# B&R Automation Studio project warcabot
Automation Studio 6.7.0.187; technology packages: mappCockpit 6.7.0, mappMotion 6.7.2, mappServices 6.7.1, mappView 6.7.0, mappVision 6.7.0, OpcUaCs 6.7.0

## Configuration Config1

CPU 5APC3100.KBU1-000, AutomationRuntime 6.7.6, Build 11.3.0

### Task classes (Cpu.sw)
```
Cyclic#4:
  Program <- Programs.Motion.Program.prg
  TestOpcua <- Programs.TestOpcua.prg
Libraries: McBase, MpRobotics, McAxGroup, McPathGen, MpAxis, runtime, CoTrace, McAxis, McAcpAx, McAcpPar, AsZip, FileIO, sys_lib, AsBrStr, MpBase, McProgInt, astime, ViBase, AsARCfg, powerlnk, AsEPL, AsIO, AsTCP, DataObj, ArSsl
```

### Hardware
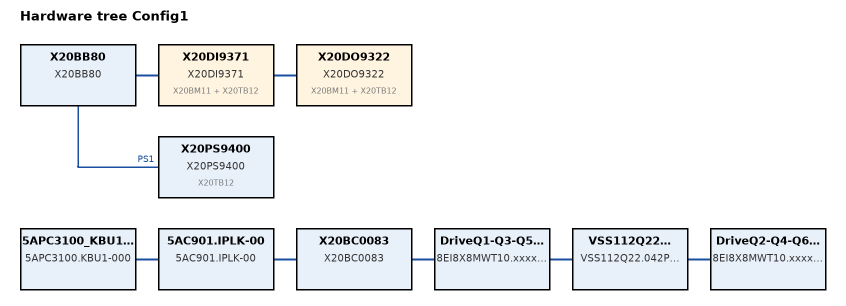
```
5AC901.IPLK-00 : 5AC901.IPLK-00 v2.1.0.0  [SL -> 5APC3100_KBU1_000.SL2]
  Connector IF1:
    MtuSize = 1500
    Channel1
    ChannelID1 = McAcpBroadcast
    ChannelType1 = OCTET[192]
    InternetAddress = 192.168.200.240
    SubnetMask = 255.255.255.0
  Supervision = off
5APC3100_KBU1_000 : 5APC3100.KBU1-000 v2.3.1.0
  Connector IF3:
    AssignedOperatingSystem = ARemb
    ActivateDevice = 1
    Mode = Manual
    InternetAddress = 192.168.0.11
    SubnetMask = 255.255.255.0
    ActivateSnmp = 2
  Connector IF4:
    AssignedOperatingSystem = ARemb
    ActivateDevice = 1
    Mode = DHCPServer
    InternetAddress = 192.168.1.11
    SubnetMask = 255.255.255.0
    Lease1
    LeaseName1 = Test
    LeaseStartAddress1 = 192.168.1.12
    LeaseStopAddress1 = 192.168.1.15
    LeaseSubnetMask1 = 255.255.255.0
    ActivateSnmp = 2
  Connector IF5:
    AssignedOperatingSystem = ARemb
  Connector IF6:
    AssignedOperatingSystem = ARemb
  Connector IF7:
    AssignedOperatingSystem = ARemb
  Connector IF8:
    AssignedOperatingSystem = ARemb
  ConfigurationID = warcabot_Config1
  Simulation = 1
  RemMemDevice = PCI.2.IPLK.SRAM
  RemMemSize = 1000
  PermanentPvSize = 500
  TimerDeviceType = EPLX2X
  TimerDevice = 5AC901.IPLK-00.IF1
  TaskClassIdleTime = 2000
  Cyclic1Duration = 2000
  Cyclic1Tolerance = 0
  FileDevice1
  FileDeviceName1 = USER
  FileDevicePath1 = USER_PATH
  FileDevice2
  FileDeviceName2 = CNC_PrgDir
  FileDevicePath2 = USER_PATH\Programs
  FileDevice3
  FileDeviceName3 = SG
  FileDevicePath3 = USER_PATH\SavedGames
  FileDevice4
  FileDeviceName4 = AH
  FileDevicePath4 = USER_PATH\AlarmHistory
  FileDevice5
  FileDeviceName5 = AUDIT
  FileDevicePath5 = USER_PATH\Audit
  FileDevice6
  FileDeviceName6 = REPORT
  FileDevicePath6 = USER_PATH\Report
  FileDevice7
  FileDeviceName7 = CF
  FileDevicePath7 = USER_PATH
  ActivateFtpServer = 1
  FtpAuthenticationType = FtpRoles
  FtpRole1
  FtpRoleName1 = Administraotr
  FTPRoleAccessRight1 = 0
  ActivateWebServer = 1
  WebServerProtocol = 1
  ActivateSdm = 1
  Authentication = 0
DriveQ1-Q3-Q5_Racer3_1 : 8EI8X8MWT10.xxxx-1 v2.4.0.0 (NodeNumber=2)  [PLK1 -> X20BC0083.PLK2 [Cable Type=PowerlinkCable, Length=10, Version=1.0.0.3]; PLK2 -> VSS112Q22.042P-000.PLK1 [Cable Type=PowerlinkCable, Length=10, Version=1.0.0.3]]
  DriveConfiguration/Encoder/EncoderX41:
    InterfaceType = EnDat
  DriveConfiguration/Encoder/EncoderX42:
    InterfaceType = EnDat
  DriveConfiguration/Encoder/EncoderX43:
    InterfaceType = EnDat
  DriveConfiguration/Channel[1]/RealAxis:
    AxisReference = gAxisQ1_Racer3_1
  DriveConfiguration/Channel[1]/RealAxis/MechanicalElements/Gearbox:
    Input = 81818
    Output = 1000
  DriveConfiguration/Channel[1]/RealAxis/MechanicalElements/RotaryToLinearTransformation:
    ReferenceDistance = 360
  DriveConfiguration/Channel[1]/RealAxis/Controller:
    Mode = PositionControllerWithTorqueFeedForward
  DriveConfiguration/Channel[1]/RealAxis/Controller/Mode/Position:
    ProportionalGain = 75
  DriveConfiguration/Channel[1]/RealAxis/Controller/Mode/Speed:
    FilterTime = 0.0008
  DriveConfiguration/Channel[1]/RealAxis/Controller/Mode:
    FeedForward = CyclicValueFromAxesGroup
  DriveConfiguration/Channel[1]/RealAxis/Homing:
    Mode = RestorePosition
    RestorePositionVariable = ::AxisRestorePos0
  DriveConfiguration/Channel[1]/RealAxis/MovementErrorLimits:
    PositionError = 1
  DriveConfiguration/Channel[1]/RealAxis:
    JerkFilter = Used
  DriveConfiguration/Channel[1]/RealAxis/JerkFilter:
    JerkTime = 0.01
  DriveConfiguration/Channel[1]/RealAxis/AxisFeatures:
    FeatureRef[1] = Feature_Brake_Racer3_1
  DriveConfiguration/Channel[2]/RealAxis:
    AxisReference = gAxisQ3_Racer3_1
  DriveConfiguration/Channel[2]/RealAxis/MechanicalElements/Gearbox:
    Input = 72
  DriveConfiguration/Channel[2]/RealAxis/MechanicalElements/RotaryToLinearTransformation:
    ReferenceDistance = 360
  DriveConfiguration/Channel[2]/RealAxis/Controller:
    Mode = PositionControllerWithTorqueFeedForward
  DriveConfiguration/Channel[2]/RealAxis/Controller/Mode/Speed:
    ProportionalGain = 1.5
    FilterTime = 0.0008
  DriveConfiguration/Channel[2]/RealAxis/Controller/Mode:
    FeedForward = CyclicValueFromAxesGroup
  DriveConfiguration/Channel[2]/RealAxis/Homing:
    Mode = RestorePosition
    RestorePositionVariable = ::AxisRestorePos2
  DriveConfiguration/Channel[2]/RealAxis/MovementErrorLimits:
    PositionError = 1
  DriveConfiguration/Channel[2]/RealAxis:
    JerkFilter = Used
  DriveConfiguration/Channel[2]/RealAxis/JerkFilter:
    JerkTime = 0.01
  DriveConfiguration/Channel[2]/RealAxis/AxisFeatures:
    FeatureRef[1] = Feature_Brake_Racer3_1
  DriveConfiguration/Channel[3]/RealAxis:
    AxisReference = gAxisQ5_Racer3_1
  DriveConfiguration/Channel[3]/RealAxis/MechanicalElements/Gearbox:
    Input = 612
    Output = 10
  DriveConfiguration/Channel[3]/RealAxis/MechanicalElements/RotaryToLinearTransformation:
    ReferenceDistance = 360
  DriveConfiguration/Channel[3]/RealAxis/Controller:
    Mode = PositionControllerWithTorqueFeedForward
  DriveConfiguration/Channel[3]/RealAxis/Controller/Mode/Position:
    ProportionalGain = 200
  DriveConfiguration/Channel[3]/RealAxis/Controller/Mode/Speed:
    ProportionalGain = 1.5
    FilterTime = 0.0008
  DriveConfiguration/Channel[3]/RealAxis/Controller/Mode:
    FeedForward = CyclicValueFromAxesGroup
  DriveConfiguration/Channel[3]/RealAxis/Homing:
    Mode = RestorePosition
    RestorePositionVariable = ::AxisRestorePos4
  DriveConfiguration/Channel[3]/RealAxis/MovementErrorLimits:
    PositionError = 1
  DriveConfiguration/Channel[3]/RealAxis:
    JerkFilter = Used
  DriveConfiguration/Channel[3]/RealAxis/JerkFilter:
    JerkTime = 0.01
  DriveConfiguration/Channel[3]/RealAxis/AxisFeatures:
    FeatureRef[1] = Feature_Brake_Racer3_1
DriveQ2-Q4-Q6_Racer3_1 : 8EI8X8MWT10.xxxx-1 v2.4.0.0 (NodeNumber=3)  [PLK1 -> VSS112Q22.042P-000.PLK2 [Cable Type=PowerlinkCable, Length=10, Version=1.0.0.3]]
  DriveConfiguration/Encoder/EncoderX41:
    InterfaceType = EnDat
  DriveConfiguration/Encoder/EncoderX42:
    InterfaceType = EnDat
  DriveConfiguration/Encoder/EncoderX43:
    InterfaceType = EnDat
  DriveConfiguration/Channel[1]/RealAxis:
    AxisReference = gAxisQ2_Racer3_1
  DriveConfiguration/Channel[1]/RealAxis/MechanicalElements/Gearbox:
    Input = 80
  DriveConfiguration/Channel[1]/RealAxis/MechanicalElements/RotaryToLinearTransformation:
    ReferenceDistance = 360
  DriveConfiguration/Channel[1]/RealAxis/Controller:
    Mode = PositionControllerWithTorqueFeedForward
  DriveConfiguration/Channel[1]/RealAxis/Controller/Mode/Speed:
    FilterTime = 0.0008
  DriveConfiguration/Channel[1]/RealAxis/Controller/Mode:
    FeedForward = CyclicValueFromAxesGroup
  DriveConfiguration/Channel[1]/RealAxis/Homing:
    Mode = RestorePosition
    RestorePositionVariable = ::AxisRestorePos1
  DriveConfiguration/Channel[1]/RealAxis/MovementErrorLimits:
    PositionError = 1
  DriveConfiguration/Channel[1]/RealAxis:
    JerkFilter = Used
  DriveConfiguration/Channel[1]/RealAxis/JerkFilter:
    JerkTime = 0.01
  DriveConfiguration/Channel[1]/RealAxis/AxisFeatures:
    FeatureRef[1] = Feature_Brake_Racer3_1
  DriveConfiguration/Channel[2]/RealAxis:
    AxisReference = gAxisQ4_Racer3_1
  DriveConfiguration/Channel[2]/RealAxis/MechanicalElements/Gearbox:
    Input = 612
    Output = 10
  DriveConfiguration/Channel[2]/RealAxis/MechanicalElements/RotaryToLinearTransformation:
    ReferenceDistance = 360
  DriveConfiguration/Channel[2]/RealAxis/Controller:
    Mode = PositionControllerWithTorqueFeedForward
  DriveConfiguration/Channel[2]/RealAxis/Controller/Mode/Position:
    ProportionalGain = 100
  DriveConfiguration/Channel[2]/RealAxis/Controller/Mode/Speed:
    FilterTime = 0.0008
  DriveConfiguration/Channel[2]/RealAxis/Controller/Mode:
    FeedForward = CyclicValueFromAxesGroup
  DriveConfiguration/Channel[2]/RealAxis/Homing:
    Mode = RestorePosition
    RestorePositionVariable = ::AxisRestorePos3
  DriveConfiguration/Channel[2]/RealAxis/MovementErrorLimits:
    PositionError = 1
  DriveConfiguration/Channel[2]/RealAxis:
    JerkFilter = Used
  DriveConfiguration/Channel[2]/RealAxis/JerkFilter:
    JerkTime = 0.01
  DriveConfiguration/Channel[2]/RealAxis/AxisFeatures:
    FeatureRef[1] = Feature_Brake_Racer3_1
  DriveConfiguration/Channel[3]/RealAxis:
    AxisReference = gAxisQ6_Racer3_1
  DriveConfiguration/Channel[3]/RealAxis/MechanicalElements/Gearbox:
    Input = 40
  DriveConfiguration/Channel[3]/RealAxis/MechanicalElements/RotaryToLinearTransformation:
    ReferenceDistance = 360
  DriveConfiguration/Channel[3]/RealAxis/Controller:
    Mode = PositionControllerWithTorqueFeedForward
  DriveConfiguration/Channel[3]/RealAxis/Controller/Mode/Position:
    ProportionalGain = 200
  DriveConfiguration/Channel[3]/RealAxis/Controller/Mode/Speed:
    ProportionalGain = 1.5
    FilterTime = 0.0008
  DriveConfiguration/Channel[3]/RealAxis/Controller/Mode:
    FeedForward = CyclicValueFromAxesGroup
  DriveConfiguration/Channel[3]/RealAxis/Homing:
    Mode = RestorePosition
    RestorePositionVariable = ::AxisRestorePos5
  DriveConfiguration/Channel[3]/RealAxis/MovementErrorLimits:
    PositionError = 1
  DriveConfiguration/Channel[3]/RealAxis:
    JerkFilter = Used
  DriveConfiguration/Channel[3]/RealAxis/JerkFilter:
    JerkTime = 0.01
  DriveConfiguration/Channel[3]/RealAxis/AxisFeatures:
    FeatureRef[1] = Feature_Brake_Racer3_1
VSS112Q22.042P-000 : VSS112Q22.042P-000 v1.11.0.929 (NodeNumber=4)  [PLK1 -> DriveQ1-Q3-Q5_Racer3_1.PLK2 [Cable Type=PowerlinkCable, Length=10, Version=1.0.0.3]; PLK2 -> DriveQ2-Q4-Q6_Racer3_1.PLK1 [Cable Type=PowerlinkCable, Length=10, Version=1.0.0.3]]
  VisionConfig = gCamera
X20BB80 : X20BB80 v1.1.0.0
X20BC0083 : X20BC0083 v2.17.0.0 (NodeNumber=1)  [PLK1 -> 5AC901.IPLK-00.IF1 [Cable Type=PowerlinkCable, Length=10, Version=1.0.0.3]; PLK2 -> DriveQ1-Q3-Q5_Racer3_1.PLK1 [Cable Type=PowerlinkCable, Length=10, Version=1.0.0.3]; SL -> X20BB80.SL1]
X20BM11 : X20BM11 v1.1.0.0  [X2X1 -> X20BB80.IF1]
X20BM11_a : X20BM11 v1.1.0.0  [X2X1 -> X20BM11.X2X2]
X20DI9371 : X20DI9371 v1.6.1.0  [SS1 -> X20TB12.SS; SL -> X20BM11.SL1]
X20DO9322 : X20DO9322 v1.7.0.0  [SS1 -> X20TB12_b.SS; SL -> X20BM11_a.SL1]
X20PS9400 : X20PS9400 v1.9.0.0  [SS1 -> X20TB12_a.SS; PS -> X20BB80.PS1]
X20TB12 : X20TB12 v1.0.0.0
X20TB12_a : X20TB12 v1.0.0.0
X20TB12_b : X20TB12 v1.0.0.0
```

### Cpu.per - 5APC3100_KBU1_000/Cpu.per
```iecst
VAR_CONFIG
	AxisRestorePos0 AT %M0; (* *)
	AxisRestorePos1 AT %M72; (* *)
	AxisRestorePos2 AT %M144; (* *)
	AxisRestorePos3 AT %M216; (* *)
	AxisRestorePos4 AT %M288; (* *)
	AxisRestorePos5 AT %M360; (* *)
END_VAR
```

### IoMap.iom - 5APC3100_KBU1_000/IoMap.iom
```iecst
VAR_CONFIG
	::Program2:gCameraCtrl.Cmd.AcquireImage AT %QX."VSS112Q22.042P-000".ImageAcquisition;
	::Program2:gCameraCtrl.Status.AcquisitionReady AT %IX."VSS112Q22.042P-000".ImageAcquisitionReady;
	::Program2:gCameraCtrl.Status.ProcessingError AT %IW."VSS112Q22.042P-000".ImageProcessingError;
	::Program2:gCameraCtrl.Status.ProcessingActive AT %IX."VSS112Q22.042P-000".ImageProcessingActive;
	::gCameraAutoAdjust AT %QX."VSS112Q22.042P-000".SearchAcquisitionSettings;
	::Program2:gCameraCtrl.Status.ReadFocus AT %IW."VSS112Q22.042P-000".ReadFocus;
	::Program2:gCameraCtrl.NumResults AT %IB."VSS112Q22.042P-000".NumResults_Out_1;
	::Program2:gCameraCtrl.Pieces[1].PositionX AT %ID."VSS112Q22.042P-000".PositionX_Out_101;
	::Program2:gCameraCtrl.Pieces[1].PositionY AT %ID."VSS112Q22.042P-000".PositionY_Out_101;
	::Program2:gCameraCtrl.Pieces[1].Area AT %ID."VSS112Q22.042P-000".Area_Out_101;
	::Program2:gCameraCtrl.Pieces[1].Score AT %IB."VSS112Q22.042P-000".Score_Out_101;
	::Program2:gCameraCtrl.Cmd.Enable AT %QX."VSS112Q22.042P-000".Enable_In_1;
	::Program2:gCameraCtrl.Pieces[1].ModelNumber AT %IB."VSS112Q22.042P-000".ModelNumber_Out_101;
	::Program2:gCameraCtrl.Parameters.NumSearchMax AT %QB."VSS112Q22.042P-000".NumSearchMax_In_1;
	::Program2:gCameraCtrl.Status.ReadExposureTime AT %ID."VSS112Q22.042P-000".ReadExposureTime;
	::Program2:gCameraCtrl.Pieces[2].ModelNumber AT %IB."VSS112Q22.042P-000".ModelNumber_Out_102;
	::Program2:gCameraCtrl.Pieces[2].Score AT %IB."VSS112Q22.042P-000".Score_Out_102;
	::Program2:gCameraCtrl.Pieces[2].PositionX AT %ID."VSS112Q22.042P-000".PositionX_Out_102;
	::Program2:gCameraCtrl.Pieces[2].PositionY AT %ID."VSS112Q22.042P-000".PositionY_Out_102;
	::Program2:gCameraCtrl.Pieces[3].ModelNumber AT %IB."VSS112Q22.042P-000".ModelNumber_Out_103;
	::Program2:gCameraCtrl.Pieces[3].Score AT %IB."VSS112Q22.042P-000".Score_Out_103;
	::Program2:gCameraCtrl.Pieces[3].PositionX AT %ID."VSS112Q22.042P-000".PositionX_Out_103;
	::Program2:gCameraCtrl.Pieces[3].PositionY AT %ID."VSS112Q22.042P-000".PositionY_Out_103;
	::Program2:gCameraCtrl.Pieces[4].ModelNumber AT %IB."VSS112Q22.042P-000".ModelNumber_Out_104;
	::Program2:gCameraCtrl.Pieces[5].ModelNumber AT %IB."VSS112Q22.042P-000".ModelNumber_Out_105;
	::Program2:gCameraCtrl.Pieces[6].ModelNumber AT %IB."VSS112Q22.042P-000".ModelNumber_Out_106;
	::Program2:gCameraCtrl.Pieces[7].ModelNumber AT %IB."VSS112Q22.042P-000".ModelNumber_Out_107;
	::Program2:gCameraCtrl.Pieces[8].ModelNumber AT %IB."VSS112Q22.042P-000".ModelNumber_Out_108;
	::Program2:gCameraCtrl.Pieces[9].ModelNumber AT %IB."VSS112Q22.042P-000".ModelNumber_Out_109;
	::Program2:gCameraCtrl.Pieces[10].ModelNumber AT %IB."VSS112Q22.042P-000".ModelNumber_Out_110;
	::Program2:gCameraCtrl.Pieces[11].ModelNumber AT %IB."VSS112Q22.042P-000".ModelNumber_Out_111;
	::Program2:gCameraCtrl.Pieces[12].ModelNumber AT %IB."VSS112Q22.042P-000".ModelNumber_Out_112;
	::Program2:gCameraCtrl.Pieces[13].ModelNumber AT %IB."VSS112Q22.042P-000".ModelNumber_Out_113;
	::Program2:gCameraCtrl.Pieces[14].ModelNumber AT %IB."VSS112Q22.042P-000".ModelNumber_Out_114;
	::Program2:gCameraCtrl.Pieces[15].ModelNumber AT %IB."VSS112Q22.042P-000".ModelNumber_Out_115;
	::Program2:gCameraCtrl.Pieces[16].ModelNumber AT %IB."VSS112Q22.042P-000".ModelNumber_Out_116;
	::Program2:gCameraCtrl.Pieces[17].ModelNumber AT %IB."VSS112Q22.042P-000".ModelNumber_Out_117;
	::Program2:gCameraCtrl.Pieces[18].ModelNumber AT %IB."VSS112Q22.042P-000".ModelNumber_Out_118;
	::Program2:gCameraCtrl.Pieces[19].ModelNumber AT %IB."VSS112Q22.042P-000".ModelNumber_Out_119;
	::Program2:gCameraCtrl.Pieces[20].ModelNumber AT %IB."VSS112Q22.042P-000".ModelNumber_Out_120;
	::Program2:gCameraCtrl.Pieces[21].ModelNumber AT %IB."VSS112Q22.042P-000".ModelNumber_Out_121;
	::Program2:gCameraCtrl.Pieces[22].ModelNumber AT %IB."VSS112Q22.042P-000".ModelNumber_Out_122;
	::Program2:gCameraCtrl.Pieces[23].ModelNumber AT %IB."VSS112Q22.042P-000".ModelNumber_Out_123;
	::Program2:gCameraCtrl.Pieces[24].ModelNumber AT %IB."VSS112Q22.042P-000".ModelNumber_Out_124;
	::Program2:gCameraCtrl.Pieces[4].Score AT %IB."VSS112Q22.042P-000".Score_Out_104;
	::Program2:gCameraCtrl.Pieces[5].Score AT %IB."VSS112Q22.042P-000".Score_Out_105;
	::Program2:gCameraCtrl.Pieces[6].Score AT %IB."VSS112Q22.042P-000".Score_Out_106;
	::Program2:gCameraCtrl.Pieces[7].Score AT %IB."VSS112Q22.042P-000".Score_Out_107;
	::Program2:gCameraCtrl.Pieces[8].Score AT %IB."VSS112Q22.042P-000".Score_Out_108;
	::Program2:gCameraCtrl.Pieces[9].Score AT %IB."VSS112Q22.042P-000".Score_Out_109;
	::Program2:gCameraCtrl.Pieces[10].Score AT %IB."VSS112Q22.042P-000".Score_Out_110;
	::Program2:gCameraCtrl.Pieces[11].Score AT %IB."VSS112Q22.042P-000".Score_Out_111;
	::Program2:gCameraCtrl.Pieces[12].Score AT %IB."VSS112Q22.042P-000".Score_Out_112;
	::Program2:gCameraCtrl.Pieces[13].Score AT %IB."VSS112Q22.042P-000".Score_Out_113;
	::Program2:gCameraCtrl.Pieces[14].Score AT %IB."VSS112Q22.042P-000".Score_Out_114;
	::Program2:gCameraCtrl.Pieces[15].Score AT %IB."VSS112Q22.042P-000".Score_Out_115;
	::Program2:gCameraCtrl.Pieces[16].Score AT %IB."VSS112Q22.042P-000".Score_Out_116;
	::Program2:gCameraCtrl.Pieces[17].Score AT %IB."VSS112Q22.042P-000".Score_Out_117;
	::Program2:gCameraCtrl.Pieces[18].Score AT %IB."VSS112Q22.042P-000".Score_Out_118;
	::Program2:gCameraCtrl.Pieces[19].Score AT %IB."VSS112Q22.042P-000".Score_Out_119;
	::Program2:gCameraCtrl.Pieces[20].Score AT %IB."VSS112Q22.042P-000".Score_Out_120;
	::Program2:gCameraCtrl.Pieces[21].Score AT %IB."VSS112Q22.042P-000".Score_Out_121;
	::Program2:gCameraCtrl.Pieces[22].Score AT %IB."VSS112Q22.042P-000".Score_Out_122;
	::Program2:gCameraCtrl.Pieces[23].Score AT %IB."VSS112Q22.042P-000".Score_Out_123;
	::Program2:gCameraCtrl.Pieces[24].Score AT %IB."VSS112Q22.042P-000".Score_Out_124;
	::Program2:gCameraCtrl.Pieces[4].PositionX AT %ID."VSS112Q22.042P-000".PositionX_Out_104;
	::Program2:gCameraCtrl.Pieces[5].PositionX AT %ID."VSS112Q22.042P-000".PositionX_Out_105;
	::Program2:gCameraCtrl.Pieces[6].PositionX AT %ID."VSS112Q22.042P-000".PositionX_Out_106;
	::Program2:gCameraCtrl.Pieces[7].PositionX AT %ID."VSS112Q22.042P-000".PositionX_Out_107;
	::Program2:gCameraCtrl.Pieces[8].PositionX AT %ID."VSS112Q22.042P-000".PositionX_Out_108;
	::Program2:gCameraCtrl.Pieces[9].PositionX AT %ID."VSS112Q22.042P-000".PositionX_Out_109;
	::Program2:gCameraCtrl.Pieces[10].PositionX AT %ID."VSS112Q22.042P-000".PositionX_Out_110;
	::Program2:gCameraCtrl.Pieces[11].PositionX AT %ID."VSS112Q22.042P-000".PositionX_Out_111;
	::Program2:gCameraCtrl.Pieces[12].PositionX AT %ID."VSS112Q22.042P-000".PositionX_Out_112;
	::Program2:gCameraCtrl.Pieces[13].PositionX AT %ID."VSS112Q22.042P-000".PositionX_Out_113;
	::Program2:gCameraCtrl.Pieces[14].PositionX AT %ID."VSS112Q22.042P-000".PositionX_Out_114;
	::Program2:gCameraCtrl.Pieces[15].PositionX AT %ID."VSS112Q22.042P-000".PositionX_Out_115;
	::Program2:gCameraCtrl.Pieces[16].PositionX AT %ID."VSS112Q22.042P-000".PositionX_Out_116;
	::Program2:gCameraCtrl.Pieces[17].PositionX AT %ID."VSS112Q22.042P-000".PositionX_Out_117;
	::Program2:gCameraCtrl.Pieces[18].PositionX AT %ID."VSS112Q22.042P-000".PositionX_Out_118;
	::Program2:gCameraCtrl.Pieces[19].PositionX AT %ID."VSS112Q22.042P-000".PositionX_Out_119;
	::Program2:gCameraCtrl.Pieces[20].PositionX AT %ID."VSS112Q22.042P-000".PositionX_Out_120;
	::Program2:gCameraCtrl.Pieces[21].PositionX AT %ID."VSS112Q22.042P-000".PositionX_Out_121;
	::Program2:gCameraCtrl.Pieces[22].PositionX AT %ID."VSS112Q22.042P-000".PositionX_Out_122;
	::Program2:gCameraCtrl.Pieces[23].PositionX AT %ID."VSS112Q22.042P-000".PositionX_Out_123;
	::Program2:gCameraCtrl.Pieces[24].PositionX AT %ID."VSS112Q22.042P-000".PositionX_Out_124;
	::Program2:gCameraCtrl.Pieces[4].PositionY AT %ID."VSS112Q22.042P-000".PositionY_Out_104;
	::Program2:gCameraCtrl.Pieces[5].PositionY AT %ID."VSS112Q22.042P-000".PositionY_Out_105;
	::Program2:gCameraCtrl.Pieces[6].PositionY AT %ID."VSS112Q22.042P-000".PositionY_Out_106;
	::Program2:gCameraCtrl.Pieces[7].PositionY AT %ID."VSS112Q22.042P-000".PositionY_Out_107;
	::Program2:gCameraCtrl.Pieces[8].PositionY AT %ID."VSS112Q22.042P-000".PositionY_Out_108;
	::Program2:gCameraCtrl.Pieces[9].PositionY AT %ID."VSS112Q22.042P-000".PositionY_Out_109;
	::Program2:gCameraCtrl.Pieces[10].PositionY AT %ID."VSS112Q22.042P-000".PositionY_Out_110;
	::Program2:gCameraCtrl.Pieces[11].PositionY AT %ID."VSS112Q22.042P-000".PositionY_Out_111;
	::Program2:gCameraCtrl.Pieces[12].PositionY AT %ID."VSS112Q22.042P-000".PositionY_Out_112;
	::Program2:gCameraCtrl.Pieces[13].PositionY AT %ID."VSS112Q22.042P-000".PositionY_Out_113;
	::Program2:gCameraCtrl.Pieces[14].PositionY AT %ID."VSS112Q22.042P-000".PositionY_Out_114;
	::Program2:gCameraCtrl.Pieces[15].PositionY AT %ID."VSS112Q22.042P-000".PositionY_Out_115;
	::Program2:gCameraCtrl.Pieces[16].PositionY AT %ID."VSS112Q22.042P-000".PositionY_Out_116;
	::Program2:gCameraCtrl.Pieces[17].PositionY AT %ID."VSS112Q22.042P-000".PositionY_Out_117;
	::Program2:gCameraCtrl.Pieces[18].PositionY AT %ID."VSS112Q22.042P-000".PositionY_Out_118;
	::Program2:gCameraCtrl.Pieces[19].PositionY AT %ID."VSS112Q22.042P-000".PositionY_Out_119;
	::Program2:gCameraCtrl.Pieces[20].PositionY AT %ID."VSS112Q22.042P-000".PositionY_Out_120;
	::Program2:gCameraCtrl.Pieces[21].PositionY AT %ID."VSS112Q22.042P-000".PositionY_Out_121;
	::Program2:gCameraCtrl.Pieces[22].PositionY AT %ID."VSS112Q22.042P-000".PositionY_Out_122;
	::Program2:gCameraCtrl.Pieces[23].PositionY AT %ID."VSS112Q22.042P-000".PositionY_Out_123;
	::Program2:gCameraCtrl.Pieces[24].PositionY AT %ID."VSS112Q22.042P-000".PositionY_Out_124;
	Cyclic#1.::doMagnet AT %QX."X20DO9322".DigitalOutput05;
	::Program2:gCameraCtrl.Parameters.ExposureTime AT %QD."VSS112Q22.042P-000".ExposureTime01;
	::Program2:gCameraCtrl.Parameters.SetFocus AT %QW."VSS112Q22.042P-000".SetFocus;
	::Program2:gCameraCtrl.Parameters.GainLevel AT %QB."VSS112Q22.042P-000".GainLevel;
	::Program2:gCameraCtrl.Status.ReadGainLevel AT %IB."VSS112Q22.042P-000".ReadGainLevel;
	::Program2:gCameraCtrl.Pieces[25].ModelNumber AT %IB."VSS112Q22.042P-000".ModelNumber_Out_125;
	::Program2:gCameraCtrl.Pieces[26].ModelNumber AT %IB."VSS112Q22.042P-000".ModelNumber_Out_126;
	::Program2:gCameraCtrl.Pieces[25].Score AT %IB."VSS112Q22.042P-000".Score_Out_125;
	::Program2:gCameraCtrl.Pieces[26].Score AT %IB."VSS112Q22.042P-000".Score_Out_126;
	::Program2:gCameraCtrl.Pieces[25].PositionX AT %ID."VSS112Q22.042P-000".PositionX_Out_125;
	::Program2:gCameraCtrl.Pieces[26].PositionX AT %ID."VSS112Q22.042P-000".PositionX_Out_126;
	::Program2:gCameraCtrl.Pieces[25].PositionY AT %ID."VSS112Q22.042P-000".PositionY_Out_125;
	::Program2:gCameraCtrl.Pieces[26].PositionY AT %ID."VSS112Q22.042P-000".PositionY_Out_126;
	::Program2:gCameraCtrl.Parameters.FlashColor AT %QB."VSS112Q22.042P-000".FlashColor01;
	::Program2:gCameraCtrl.Parameters.FlashSegment AT %QB."VSS112Q22.042P-000".FlashSegment01;
END_VAR
```

### GroupConf.axesgroup - 5APC3100_KBU1_000/mappMotion/6AxesRoboArmA/GroupConf.axesgroup
```
Element gAxesGroup_Racer3_1 (Type=axesgroup)
  Type = PathGenAxesGroup
    PhysicalAxes:
      JointAxes:
        JointAxis[1]:
          AxisRef = gAxisQ1_Racer3_1
        JointAxis[2]:
          AxisRef = gAxisQ2_Racer3_1
        JointAxis[3]:
          AxisRef = gAxisQ3_Racer3_1
        JointAxis[4]:
          AxisRef = gAxisQ4_Racer3_1
        JointAxis[5]:
          AxisRef = gAxisQ5_Racer3_1
        JointAxis[6]:
          AxisRef = gAxisQ6_Racer3_1
    MechanicalSystem:
      MechSysRef = MechSys_Racer3_1
    BasicSettings:
      GeometryPlanning:
        MaxTangentialTransitionDeviation = 0.05
      TrajectoryPlanning:
        LimitCheckResolution:
          Time = 0.005
        BufferTime:
          Time = 0.050
    AxesGroupFeatures:
      FeatureRef[1] = Feature_Programs_Racer3_1
      FeatureRef[2] = Feature_FeedForward_Racer3_1
      FeatureRef[3] = Feature_Jogging_Racer3_1
      FeatureRef[4] = Feature_SharedBrakesSignals_Racer3_1
      FeatureRef[5] = Feature_WorkspaceMonitoring_Racer3_1
```

### GroupFeat.axesgroupfeature - 5APC3100_KBU1_000/mappMotion/6AxesRoboArmA/GroupFeat.axesgroupfeature
```
Element Feature_Programs_Racer3_1 (Type=axesgroupfeature)
Element Feature_FeedForward_Racer3_1 (Type=axesgroupfeature)
  Type = FeedForward
    RiseTime = 0.25
Element Feature_Jogging_Racer3_1 (Type=axesgroupfeature)
  Type = Jogging
Element Feature_SharedBrakesSignals_Racer3_1 (Type=axesgroupfeature)
  Type = SharedBrakesSignals
    BrakeComposite[1]:
      Axes:
        AxisRef[1] = gAxisQ1_Racer3_1
        AxisRef[2] = gAxisQ2_Racer3_1
        AxisRef[3] = gAxisQ3_Racer3_1
      Output:
        AxisRef = gAxisQ1_Racer3_1
    BrakeComposite[2]:
      Axes:
        AxisRef[1] = gAxisQ4_Racer3_1
        AxisRef[2] = gAxisQ5_Racer3_1
        AxisRef[3] = gAxisQ6_Racer3_1
      Output:
        AxisRef = gAxisQ4_Racer3_1
Element Feature_WorkspaceMonitoring_Racer3_1 (Type=axesgroupfeature)
  Type = WorkspaceMonitoring
    WorkspaceRef = Workspace_1
    SelfCollisionDetection = Enabled
Element Feature_Monitoring_Racer3_2 (Type=axesgroupfeature)
  Type = MonitoringElements
    SingleElements:
      SingleElement[1] = WorkspaceMonitoring
        Level = ::WorkspaceMonitor
```

### MechSys.mechanicalsystem - 5APC3100_KBU1_000/mappMotion/6AxesRoboArmA/MechSys.mechanicalsystem
```
Element MechSys_Racer3_1 (Type=mechanicalsystem)
  Type = 6AxesRoboarm
    Subtype = 6AxesRoboarmB
      Description:
        Dimensions:
          TranslationFromBaseToQ1IsReadOnly = 1
          TranslationFromQ1ToQ2IsReadOnly = 1
          TranslationFromQ1ToQ2:
            X = 50.0
            Z = 365.0
          TranslationFromQ2ToQ3IsReadOnly = 1
          TranslationFromQ2ToQ3:
            Z = 270.0
          TranslationFromQ3ToQ4IsReadOnly = 1
          TranslationFromQ3ToQ4:
            X = -50.0
          TranslationFromQ4ToQ5IsReadOnly = 1
          TranslationFromQ4ToQ5:
            Z = 305.94
          TranslationFromQ5ToQ6IsReadOnly = 1
          TranslationFromQ6ToFlange:
            Z = 120
        Offsets:
          JointAxisIsReadOnly = 1
          JointAxis[1]
          JointAxis[2]
          JointAxis[3]
          JointAxis[4]
          JointAxis[5]
          JointAxis[6]
        CountDirections:
          JointAxisIsReadOnly = 1
          JointAxis[1] = Inverse
          JointAxis[2]
          JointAxis[3] = Inverse
          JointAxis[4] = Inverse
          JointAxis[5]
          JointAxis[6] = Inverse
      InternalDynamicModel = Used
        TypeIsReadOnly = 1
        Type = Comau Racer 3
        Row[1]:
          Value = 4
          Unit = 
          Description = TRF_DYN11D_typ
        Row[2]:
          Index = 1
          Value = 0
          Unit = 
          Description = 
        Row[3]:
          Index = 2
          Value = 0
          Unit = 
          Description = 
        Row[4]:
          Index = 3
          Value = 0.99502
          Unit = kgm^2
          Description = m1*rc1x^2+m1*rc1y^2+Jzz1+(0.0025)*m2+m2*rc2y^2+(0.5)*Jxx2+(-0.5)*Jyy2+(0.5)*Jzz2+(0.0025)*m3+m3*rc3y^2+(0.5)*Jxx3+(-0.5)*Jyy3+(0.5)*Jzz3+(0.0025)*m4+(0.0025)*m5+(0.0025)*m6+(6694.1851)*JDrive1+(-3200)*JDrive2
        Row[5]:
          Index = 4
          Value = 0
          Unit = 
          Description = 
        Row[6]:
          Index = 5
          Value = 0
          Unit = 
          Description = 
        Row[7]:
          Index = 6
          Value = 0
          Unit = 
          Description = 
        Row[8]:
          Index = 7
          Value = -0.0079739
          Unit = kgm
          Description = m2*rc2x
        Row[9]:
          Index = 8
          Value = 0
          Unit = 
          Description = 
        Row[10]:
          Index = 9
          Value = 3.2569
          Unit = kgm
          Description = m2*rc2z+(0.27)*m3+(0.27)*m4+(0.27)*m5+(0.27)*m6
        Row[11]:
          Index = 10
          Value = -0.01529
          Unit = kgm^2
          Description = m2*rc2x*rc2y
        Row[12]:
          Index = 11
          Value = 0.018218
          Unit = kgm^2
          Description = m2*rc2y*rc2z+(0.27)*m3*rc3y
        Row[13]:
          Index = 12
          Value = -0.027
          Unit = kgm^2
          Description = m2*rc2x*rc2z
        Row[14]:
          Index = 13
          Value = 0.23153
          Unit = kgm^2
          Description = m2*rc2x^2+(-0.5)*Jxx2+(0.5)*Jyy2+(0.5)*Jzz2+(3200)*JDrive2
        Row[15]:
          Index = 14
          Value = 0
          Unit = 
          Description = 
        Row[16]:
          Index = 15
          Value = 1.1014
          Unit = kgm^2
          Description = m2*rc2z^2+(0.5)*Jxx2+(0.5)*Jyy2+(-0.5)*Jzz2+(0.0729)*m3+(0.0729)*m4+(0.0729)*m5+(0.0729)*m6+(3200)*JDrive2
        Row[17]:
          Index = 16
          Value = 0
          Unit = 
          Description = 
        Row[18]:
          Index = 17
          Value = 0
          Unit = 
          Description = 
        Row[19]:
          Index = 18
          Value = 0
          Unit = 
          Description = 
        Row[20]:
          Index = 19
          Value = 0
          Unit = 
          Description = 
        Row[21]:
          Index = 20
          Value = -0.32261
          Unit = kgm
          Description = m3*rc3x+(-0.05)*m4+(-0.05)*m5+(-0.05)*m6
        Row[22]:
          Index = 21
          Value = 0
          Unit = 
          Description = 
        Row[23]:
          Index = 22
          Value = 1.1289
          Unit = kgm
          Description = m3*rc3z+m4*rc4z+(0.30594)*m5+(0.30594)*m6
        Row[24]:
          Index = 23
          Value = -0.0059741
          Unit = kgm^2
          Description = m3*rc3x*rc3y
        Row[25]:
          Index = 24
          Value = 0.048102
          Unit = kgm^2
          Description = m3*rc3y*rc3z
        Row[26]:
          Index = 25
          Value = -0.049555
          Unit = kgm^2
          Description = m3*rc3x*rc3z+(-0.05)*m4*rc4z+(-0.015297)*m5+(-0.015297)*m6
        Row[27]:
          Index = 26
          Value = -0.026241
          Unit = kgm^2
          Description = m3*rc3x^2+(-0.5)*Jxx3+(0.5)*Jyy3+(0.5)*Jzz3+(0.0025)*m4+(0.0025)*m5+(0.0025)*m6
        Row[28]:
          Index = 27
          Value = 0
          Unit = 
          Description = 
        Row[29]:
          Index = 28
          Value = 0.21145
          Unit = kgm^2
          Description = m3*rc3z^2+(0.5)*Jxx3+(0.5)*Jyy3+(-0.5)*Jzz3+m4*rc4z^2+(0.5)*Jxx4+(0.5)*Jyy4+(-0.5)*Jzz4+(0.093599)*m5+(0.093599)*m6
        Row[30]:
          Index = 29
          Value = 0
          Unit = 
          Description = 
        Row[31]:
          Index = 30
          Value = 0
          Unit = 
          Description = 
        Row[32]:
          Index = 31
          Value = 0
          Unit = 
          Description = 
        Row[33]:
          Index = 32
          Value = 0
          Unit = 
          Description = 
        Row[34]:
          Index = 33
          Value = -0.0056373
          Unit = kgm
          Description = m4*rc4x
        Row[35]:
          Index = 34
          Value = 0.011806
          Unit = kgm
          Description = m4*rc4y+m5*rc5y
        Row[36]:
          Index = 35
          Value = 0
          Unit = 
          Description = 
        Row[37]:
          Index = 36
          Value = -0.0071612
          Unit = kgm^2
          Description = m4*rc4x*rc4y
        Row[38]:
          Index = 37
          Value = -0.00018934
          Unit = kgm^2
          Description = m4*rc4y*rc4z+(0.30594)*m5*rc5y
        Row[39]:
          Index = 38
          Value = 0.002269
          Unit = kgm^2
          Description = m4*rc4x*rc4z
        Row[40]:
          Index = 39
          Value = -0.0073563
          Unit = kgm^2
          Description = m4*rc4x^2+(-0.5)*Jxx4+(0.5)*Jyy4+(0.5)*Jzz4
        Row[41]:
          Index = 40
          Value = -0.00050442
          Unit = kgm^2
          Description = m4*rc4y^2+(0.5)*Jxx4+(-0.5)*Jyy4+(0.5)*Jzz4+m5*rc5y^2+(0.5)*Jxx5+(-0.5)*Jyy5+(0.5)*Jzz5
        Row[42]:
          Index = 41
          Value = 0
          Unit = 
          Description = 
        Row[43]:
          Index = 42
          Value = 0
          Unit = 
          Description = 
        Row[44]:
          Index = 43
          Value = 0
          Unit = 
          Description = 
        Row[45]:
          Index = 44
          Value = 0
          Unit = 
          Description = 
        Row[46]:
          Index = 45
          Value = 0
          Unit = 
          Description = 
        Row[47]:
          Index = 46
          Value = -0.0030729
          Unit = kgm
          Description = m5*rc5x
        Row[48]:
          Index = 47
          Value = 0
          Unit = 
          Description = 
        Row[49]:
          Index = 48
          Value = 0.0086628
          Unit = kgm
          Description = m5*rc5z+m6*rc6z
        Row[50]:
          Index = 49
          Value = 5.0384e-05
          Unit = kgm^2
          Description = m5*rc5x*rc5y
        Row[51]:
          Index = 50
          Value = 0.004449
          Unit = kgm^2
          Description = m5*rc5y*rc5z
        Row[52]:
          Index = 51
          Value = 0.00094987
          Unit = kgm^2
          Description = m5*rc5x*rc5z
        Row[53]:
          Index = 52
          Value = -0.0039698
          Unit = kgm^2
          Description = m5*rc5x^2+(-0.5)*Jxx5+(0.5)*Jyy5+(0.5)*Jzz5
        Row[54]:
          Index = 53
          Value = 0
          Unit = 
          Description = 
        Row[55]:
          Index = 54
          Value = -0.0023413
          Unit = kgm^2
          Description = m5*rc5z^2+(0.5)*Jxx5+(0.5)*Jyy5+(-0.5)*Jzz5+m6*rc6z^2+(0.5)*Jxx6+(0.5)*Jyy6+(-0.5)*Jzz6
        Row[56]:
          Index = 55
          Value = 0
          Unit = 
          Description = 
        Row[57]:
          Index = 56
          Value = 0
          Unit = 
          Description = 
        Row[58]:
          Index = 57
          Value = 0
          Unit = 
          Description = 
        Row[59]:
          Index = 58
          Value = 0
          Unit = 
          Description = 
        Row[60]:
          Index = 59
          Value = 0.00052765
          Unit = kgm
          Description = m6*rc6x
        Row[61]:
          Index = 60
          Value = -0.0030867
          Unit = kgm
          Description = m6*rc6y
        Row[62]:
          Index = 61
          Value = 0
          Unit = 
          Description = 
        Row[63]:
          Index = 62
          Value = 5.0962e-05
          Unit = kgm^2
          Description = m6*rc6x*rc6y
        Row[64]:
          Index = 63
          Value = -0.0015762
          Unit = kgm^2
          Description = m6*rc6y*rc6z
        Row[65]:
          Index = 64
          Value = 0.0005846
          Unit = kgm^2
          Description = m6*rc6x*rc6z
        Row[66]:
          Index = 65
          Value = 0.00067399
          Unit = kgm^2
          Description = m6*rc6x^2+(-0.5)*Jxx6+(0.5)*Jyy6+(0.5)*Jzz6
        Row[67]:
          Index = 66
          Value = 0.0013929
          Unit = kgm^2
          Description = m6*rc6y^2+(0.5)*Jxx6+(-0.5)*Jyy6+(0.5)*Jzz6
        Row[68]:
          Index = 67
          Value = 0
          Unit = 
          Description = 
        Row[69]:
          Index = 68
          Value = 0
          Unit = 
          Description = 
        Row[70]:
          Index = 69
          Value = 0
          Unit = 
          Description = 
        Row[71]:
          Index = 70
          Value = 0
          Unit = 
          Description = 
        Row[72]:
          Index = 71
          Value = 0
          Unit = 
          Description = mTool
        Row[73]:
          Index = 72
          Value = 0
          Unit = 
          Description = mTool*rcToolx
        Row[74]:
          Index = 73
          Value = 0
          Unit = 
          Description = mTool*rcTooly
        Row[75]:
          Index = 74
          Value = 0
          Unit = 
          Description = mTool*rcToolz
        Row[76]:
          Index = 75
          Value = 0
          Unit = 
          Description = mTool*rcToolx*rcTooly
        Row[77]:
          Index = 76
          Value = 0
          Unit = 
          Description = mTool*rcTooly*rcToolz
        Row[78]:
          Index = 77
          Value = 0
          Unit = 
          Description = mTool*rcToolx*rcToolz
        Row[79]:
          Index = 78
          Value = 0
          Unit = 
          Description = mTool*rcToolx^2
        Row[80]:
          Index = 79
          Value = 0
          Unit = 
          Description = mTool*rcTooly^2
        Row[81]:
          Index = 80
          Value = 0
          Unit = 
          Description = mTool*rcToolz^2
        Row[82]:
          Index = 81
          Value = 0
          Unit = 
          Description = JxxTool
        Row[83]:
          Index = 82
          Value = 0
          Unit = 
          Description = JyyTool
        Row[84]:
          Index = 83
          Value = 0
          Unit = 
          Description = JzzTool
        Row[85]:
          Index = 84
          Value = 0
          Unit = 
          Description = 
        Row[86]:
          Index = 85
          Value = 0
          Unit = 
          Description = 
        Row[87]:
          Index = 86
          Value = 9.8824e-05
          Unit = kgm^2
          Description = JDrive3
        Row[88]:
          Index = 87
          Value = 5.2689e-05
          Unit = kgm^2
          Description = JDrive4
        Row[89]:
          Index = 88
          Value = 5.129e-05
          Unit = kgm^2
          Description = JDrive5
        Row[90]:
          Index = 89
          Value = 5.2318e-05
          Unit = kgm^2
          Description = JDrive6
        Row[91]:
          Index = 90
          Value = 4.1946
          Unit = Nms
          Description = dV1
        Row[92]:
          Index = 91
          Value = 7.0888
          Unit = Nms
          Description = dV2
        Row[93]:
          Index = 92
          Value = 3.1195
          Unit = Nms
          Description = dV3
        Row[94]:
          Index = 93
          Value = 1.481
          Unit = Nms
          Description = dV4
        Row[95]:
          Index = 94
          Value = 1.1989
          Unit = Nms
          Description = dV5
        Row[96]:
          Index = 95
          Value = 0.67577
          Unit = Nms
          Description = dV6
        Row[97]:
          Index = 96
          Value = 25.5954
          Unit = Nm
          Description = dC1
        Row[98]:
          Index = 97
          Value = 14.3239
          Unit = Nm
          Description = dC2
        Row[99]:
          Index = 98
          Value = 7.6123
          Unit = Nm
          Description = dC3
        Row[100]:
          Index = 99
          Value = 7.9035
          Unit = Nm
          Description = dC4
        Row[101]:
          Index = 100
          Value = 3.5858
          Unit = Nm
          Description = dC5
        Row[102]:
          Index = 101
          Value = 5.2501
          Unit = Nm
          Description = dC6
      Couplings:
        LinearCoupling[1]:
          SourceAxisIsReadOnly = 1
          SourceAxis = 5
          SourceAxisUnitsIsReadOnly = 1
          SourceAxisUnits = 1.0
          TargetJointAxisIsReadOnly = 1
          TargetJointAxis = 6
          TargetJointAxisUnitsIsReadOnly = 1
          TargetJointAxisUnits = 0.02
      JointAxesPositionLimits:
        JointAxis[1] = ConfigureJointAxesLimits
          LowerLimitMin = -170.0
          UpperLimitMax = 170.0
          LowerLimit = -170.0
          UpperLimit = 170.0
        JointAxis[2] = ConfigureJointAxesLimits
          LowerLimitMin = -95.0
          UpperLimitMax = 135.0
          LowerLimit = -95.0
          UpperLimit = 135.0
        JointAxis[3] = ConfigureJointAxesLimits
          LowerLimitMin = -155.0
          UpperLimitMax = 90.0
          LowerLimit = -155.0
          UpperLimit = 90.0
        JointAxis[4] = ConfigureJointAxesLimits
          LowerLimitMin = -200.0
          UpperLimitMax = 200.0
          LowerLimit = -200.0
          UpperLimit = 200.0
        JointAxis[5] = ConfigureJointAxesLimits
          LowerLimitMin = -125.0
          UpperLimitMax = 125.0
          LowerLimit = -125.0
          UpperLimit = 125.0
        JointAxis[6] = ConfigureJointAxesLimits
          LowerLimitMin = -2700.0
          UpperLimitMax = 2700.0
          LowerLimit = -2700.0
          UpperLimit = 2700.0
```

### AxisConf.axis - 5APC3100_KBU1_000/mappMotion/AxisConf.axis
```
Element gAxisQ1_Racer3_1 (Type=axis)
  BaseTypeIsReadOnly = 1
  BaseType = RotaryBounded
    MeasurementUnitIsReadOnly = 1
    MeasurementResolutionIsReadOnly = 1
    MeasurementResolution = 0.001
    CountDirection = Inverse
  MovementLimitsIsReadOnly = 1
  MovementLimits = InternalForPathControlledAxis
    Position:
      LowerLimitMin = -170.0
      UpperLimitMax = 170.0
      LowerLimit = -170.0
      UpperLimit = 170.0
    VelocityIsReadOnly = 1
    Velocity:
      VelocityMax = 420.0
      Velocity = 420.0
    AccelerationIsReadOnly = 1
    Acceleration:
      AccelerationMax = 1100.0
      Acceleration = 1100.0
    DecelerationIsReadOnly = 1
    Deceleration:
      DecelerationMax = 1100.0
      Deceleration = 1100.0
    JerkIsReadOnly = 1
    Jerk = Basic
      Jerk = 11000.0
    TorqueIsReadOnly = 1
Element gAxisQ2_Racer3_1 (Type=axis)
  BaseTypeIsReadOnly = 1
  BaseType = RotaryBounded
    MeasurementUnitIsReadOnly = 1
    MeasurementResolutionIsReadOnly = 1
    MeasurementResolution = 0.001
    CountDirectionIsReadOnly = 1
  MovementLimitsIsReadOnly = 1
  MovementLimits = InternalForPathControlledAxis
    Position:
      LowerLimitMin = -95.0
      UpperLimitMax = 135.0
      LowerLimit = -95.0
      UpperLimit = 135.0
    VelocityIsReadOnly = 1
    Velocity:
      VelocityMax = 450.0
      Velocity = 450.0
    AccelerationIsReadOnly = 1
    Acceleration:
      AccelerationMax = 750.0
      Acceleration = 750.0
    DecelerationIsReadOnly = 1
    Deceleration:
      DecelerationMax = 750.0
      Deceleration = 750.0
    JerkIsReadOnly = 1
    Jerk = Basic
      Jerk = 7500.0
    TorqueIsReadOnly = 1
Element gAxisQ3_Racer3_1 (Type=axis)
  BaseTypeIsReadOnly = 1
  BaseType = RotaryBounded
    MeasurementUnitIsReadOnly = 1
    MeasurementResolutionIsReadOnly = 1
    MeasurementResolution = 0.001
    CountDirectionIsReadOnly = 1
    CountDirection = Inverse
  MovementLimitsIsReadOnly = 1
  MovementLimits = InternalForPathControlledAxis
    Position:
      LowerLimitMin = -155.0
      UpperLimitMax = 90.0
      LowerLimit = -155.0
      UpperLimit = 90.0
    VelocityIsReadOnly = 1
    Velocity:
      VelocityMax = 480.0
      Velocity = 480.0
    AccelerationIsReadOnly = 1
    Acceleration:
      AccelerationMax = 1250.0
      Acceleration = 1250.0
    DecelerationIsReadOnly = 1
    Deceleration:
      DecelerationMax = 1250.0
      Deceleration = 1250.0
    JerkIsReadOnly = 1
    Jerk = Basic
      Jerk = 12500.0
    TorqueIsReadOnly = 1
Element gAxisQ4_Racer3_1 (Type=axis)
  BaseTypeIsReadOnly = 1
  BaseType = RotaryBounded
    MeasurementUnitIsReadOnly = 1
    MeasurementResolutionIsReadOnly = 1
    MeasurementResolution = 0.001
    CountDirectionIsReadOnly = 1
  MovementLimitsIsReadOnly = 1
  MovementLimits = InternalForPathControlledAxis
    Position:
      LowerLimitMin = -200.0
      UpperLimitMax = 200.0
      LowerLimit = -200.0
      UpperLimit = 200.0
    VelocityIsReadOnly = 1
    Velocity:
      VelocityMax = 600.0
      Velocity = 600.0
    AccelerationIsReadOnly = 1
    Acceleration:
      AccelerationMax = 1200.0
      Acceleration = 1200.0
    DecelerationIsReadOnly = 1
    Deceleration:
      DecelerationMax = 1200.0
      Deceleration = 1200.0
    JerkIsReadOnly = 1
    Jerk = Basic
      Jerk = 12000.0
    TorqueIsReadOnly = 1
Element gAxisQ5_Racer3_1 (Type=axis)
  BaseTypeIsReadOnly = 1
  BaseType = RotaryBounded
    MeasurementUnitIsReadOnly = 1
    MeasurementResolutionIsReadOnly = 1
    MeasurementResolution = 0.001
    CountDirectionIsReadOnly = 1
  MovementLimitsIsReadOnly = 1
  MovementLimits = InternalForPathControlledAxis
    Position:
      LowerLimitMin = -125.0
      UpperLimitMax = 125.0
      LowerLimit = -125.0
      UpperLimit = 125.0
    VelocityIsReadOnly = 1
    Velocity:
      VelocityMax = 600.0
      Velocity = 600.0
    AccelerationIsReadOnly = 1
    Acceleration:
      AccelerationMax = 1200.0
      Acceleration = 1200.0
    DecelerationIsReadOnly = 1
    Deceleration:
      DecelerationMax = 1200.0
      Deceleration = 1200.0
    JerkIsReadOnly = 1
    Jerk = Basic
      Jerk = 12000.0
    TorqueIsReadOnly = 1
Element gAxisQ6_Racer3_1 (Type=axis)
  BaseTypeIsReadOnly = 1
  BaseType = RotaryBounded
    MeasurementUnitIsReadOnly = 1
    MeasurementResolutionIsReadOnly = 1
    MeasurementResolution = 0.001
    CountDirectionIsReadOnly = 1
  MovementLimitsIsReadOnly = 1
  MovementLimits = InternalForPathControlledAxis
    Position:
      LowerLimitMin = -2700.0
      UpperLimitMax = 2700.0
      LowerLimit = -2700.0
      UpperLimit = 2700.0
    VelocityIsReadOnly = 1
    Velocity:
      VelocityMax = 875.0
      Velocity = 875.0
    AccelerationIsReadOnly = 1
    Acceleration:
      AccelerationMax = 1800.0
      Acceleration = 1800.0
    DecelerationIsReadOnly = 1
    Deceleration:
      DecelerationMax = 1800.0
      Deceleration = 1800.0
    JerkIsReadOnly = 1
    Jerk = Basic
      Jerk = 18000.0
    TorqueIsReadOnly = 1
```

### AxisFeat.axisfeature - 5APC3100_KBU1_000/mappMotion/AxisFeat.axisfeature
```
Element Feature_Brake_Racer3_1 (Type=axisfeature)
  Type = Brake
    BrakeControlType:
      ControlMode = External
        CommandAcceptance = Any
      ControlMonitoring = NotUsed
      MovementMonitoring = NotUsed
```

### GroupConf.axesgroup - 5APC3100_KBU1_000/mappMotion/GroupConf.axesgroup
```
Element gAxesGroup_Racer3_1 (Type=axesgroup)
  Type = PathGenAxesGroup
    PhysicalAxes:
      JointAxes:
        JointAxis[1]:
          AxisRef = gAxisQ1_Racer3_1
        JointAxis[2]:
          AxisRef = gAxisQ2_Racer3_1
        JointAxis[3]:
          AxisRef = gAxisQ3_Racer3_1
        JointAxis[4]:
          AxisRef = gAxisQ4_Racer3_1
        JointAxis[5]:
          AxisRef = gAxisQ5_Racer3_1
        JointAxis[6]:
          AxisRef = gAxisQ6_Racer3_1
    MechanicalSystem:
      MechSysRef = MechSys_Racer3_1
    BasicSettings:
      GeometryPlanning:
        MaxTangentialTransitionDeviation = 0.05
      TrajectoryPlanning:
        LimitCheckResolution:
          Time = 0.005
        BufferTime:
          Time = 0.050
    AxesGroupFeatures:
      FeatureRef[1] = Feature_Programs_Racer3_1
      FeatureRef[2] = Feature_FeedForward_Racer3_1
      FeatureRef[3] = Feature_Jogging_Racer3_1
      FeatureRef[4] = Feature_SharedBrakesSignals_Racer3_1
```

### GroupFeat.axesgroupfeature - 5APC3100_KBU1_000/mappMotion/GroupFeat.axesgroupfeature
```
Element Feature_Programs_Racer3_1 (Type=axesgroupfeature)
Element Feature_FeedForward_Racer3_1 (Type=axesgroupfeature)
  Type = FeedForward
    RiseTime = 0.25
Element Feature_Jogging_Racer3_1 (Type=axesgroupfeature)
  Type = Jogging
Element Feature_SharedBrakesSignals_Racer3_1 (Type=axesgroupfeature)
  Type = SharedBrakesSignals
    BrakeComposite[1]:
      Axes:
        AxisRef[1] = gAxisQ1_Racer3_1
        AxisRef[2] = gAxisQ2_Racer3_1
        AxisRef[3] = gAxisQ3_Racer3_1
      Output:
        AxisRef = gAxisQ1_Racer3_1
    BrakeComposite[2]:
      Axes:
        AxisRef[1] = gAxisQ4_Racer3_1
        AxisRef[2] = gAxisQ5_Racer3_1
        AxisRef[3] = gAxisQ6_Racer3_1
      Output:
        AxisRef = gAxisQ4_Racer3_1
```

### AuditTrial.mpaudittrail - 5APC3100_KBU1_000/mappServices/AuditTrial.mpaudittrail
```
Element gAuditTrail (Type=mpaudittrail)
  mapp.Gen:
    Enable = TRUE
    EnableCockpit = FALSE
    EnableOpcUa = TRUE
    TaskClass = 4
    Parent
  Audit:
    Events:
      [0] = 100
      [1] = 101
      [2] = 102
      [3] = 104
      [4] = 400
      [5] = 700
      [6] = 600
      [7] = 150
      [8] = 103
    EventFilter
    Memory = 0
      Size = 200
      Interval = 60
      BufferSize = 10
    TextSource:
      DisplayFormat = {&evtime[TIME=%c]} {&ev}
      ExportFormat = Same
    Archive = Off
    Export:
      RawData = FALSE
      FileType = 0
      Encrypt = FALSE
      PassPhrase
  Alarms = MpAlarmX
    mapp.AlarmX.Core.Configuration:
      [0]:
        Name = ArchiveAvailable
        Message = {$BR/mapp/MpAuditTrail/Alarms/ArchiveAvailable}
        Code = 0
        Severity = 1
        Behavior = PersistentAlarm
          AutoReset = FALSE
          Acknowledge = 1
          Confirm = 0
          MultipleInstances = FALSE
          ReactionWhilePending = TRUE
          Async = FALSE
          DataUpdate:
            Activation:
              TimeStamp = FALSE
              Snippets = FALSE
          Recording:
            InactiveToActive = TRUE
            ActiveToInactive = FALSE
            UnacknowledgedToAcknowledged = TRUE
            AcknowledgedToUnacknowledged = TRUE
            UnconfirmedToConfirmed = TRUE
            ConfirmedToUnconfirmed = TRUE
            Update = FALSE
        Disable = FALSE
        AdditionalInformation1
        AdditionalInformation2
      [1]:
        Name = MaxArchives
        Message = {$BR/mapp/MpAuditTrail/Alarms/MaxArchives}
        Code = 0
        Severity = 1
        Behavior = EdgeAlarm
          AutoReset = TRUE
          Acknowledge = 1
          Confirm = 0
          MultipleInstances = TRUE
          ReactionWhilePending = TRUE
          Async = FALSE
          Recording:
            InactiveToActive = TRUE
            ActiveToInactive = FALSE
            UnacknowledgedToAcknowledged = TRUE
            UnconfirmedToConfirmed = TRUE
        Disable = FALSE
        AdditionalInformation1
        AdditionalInformation2
```

### ConfAlHist.mpalarmxhistory - 5APC3100_KBU1_000/mappServices/ConfAlHist.mpalarmxhistory
```
Element MpLinkgAlarmXHistory (Type=mpalarmxhistory)
  mapp.Gen:
    Enable = TRUE
    EnableCockpit = FALSE
    EnableOpcUa = FALSE
    TaskClass = 4
    Audit = TRUE
    Parent
  mapp.AlarmX.History:
    Export:
      TimeStampPattern = %Y-%m-%d %H:%M:%S:%L
      AutoExtension = TRUE
      ColumnSeparator = ,
    Memory = 0
      Size = 200
      BufferSize = 10
      Interval = 60
    Scope = 0
```

### ConfAlList.mpalarmxlist - 5APC3100_KBU1_000/mappServices/ConfAlList.mpalarmxlist
```
Element gAlarmXList (Type=mpalarmxlist)
  mapp.AlarmX.Core.Configuration:
    [0]:
      Name = MergeError
      Message = Merge się nie powiódł, wołaj Gitmastera
      Code = 0
      Severity = 1
      Behavior = EdgeAlarm
        Confirm = 0
        ReactionWhilePending = TRUE
        Retain = FALSE
        Async = FALSE
        DataUpdate:
          Activation:
            TimeStamp = FALSE
            Snippets = FALSE
        Recording:
          InactiveToActive = TRUE
          UnacknowledgedToAcknowledged = TRUE
          AcknowledgedToUnacknowledged = FALSE
          UnconfirmedToConfirmed = TRUE
          ConfirmedToUnconfirmed = FALSE
      Disable = FALSE
      InhibitPV
      AdditionalInformation1
      AdditionalInformation2
    [1]:
      Name = Test
      Message = Testowanie nocą
      Code = 1
      Severity = 1
      Behavior = LevelMonitoring
        Confirm = 0
        ReactionWhilePending = TRUE
        Recording:
          InactiveToActive = TRUE
          UnacknowledgedToAcknowledged = TRUE
          AcknowledgedToUnacknowledged = FALSE
          UnconfirmedToConfirmed = TRUE
          ConfirmedToUnconfirmed = FALSE
          Update = FALSE
        Monitoring:
          MonitoredPV = ::AlarmHisto:AlarmTest
          Exclusive = TRUE
          LowLimitEnable = Disabled
          LowLowLimitEnable = Disabled
          HighLimitEnable = Static
            Limit = 5
            LimitText
          HighHighLimitEnable = Static
            Limit = 10
            LimitText
          Settings = 0
            Delay = 0.0
            Hysteresis = 0.0
      Disable = FALSE
      InhibitPV
      AdditionalInformation1
      AdditionalInformation2
  mapp.AlarmX.Snippets:
    AutoDetect = 1
      Language
```

### Config.mpuserx - 5APC3100_KBU1_000/mappServices/Config.mpuserx
```
Element UserMgmtX (Type=mpuserx)
  mapp.Gen:
    Audit = TRUE
  UserMgmtSystem:
    UserMgmtSystemType = 0
  ServerSettings:
    Server = ADServer
      Timeout = 10
      Mapping:
        TableName
      DisplayName = username
      AdditionalUserData:
        [0] = mail
        [1] = telephoneNumber
  PasswordPolicy:
    PasswordMaxAge = 0
    PasswordExpirationNotification = 0
    PasswordHistory = 0
    PasswordChangeReq = FALSE
    PasswordCase = FALSE
    PasswordAlpha = FALSE
    PasswordSpecial = FALSE
    PasswordLength = 1
  UserAccount:
    InvalidPasswordAttempts = 3
    UserExpirationTime = 0
    AutoLogoutTime = 3600
    UserNameLength = 1
    NoDelete = FALSE
    AdminUnlockTime = 3600
    EditSameLevel = 1
  ImportExport:
    ImportUser = 2
    ImportRole = 2
    ImportUnchecked = FALSE
    FileChecksum = 2
  Users:
    DefUser#1:
      id = Admin
      name = Administroator
      lang
      measSystem = 0
    DefUser#2:
      id = User
      name = Operator
      lang
      measSystem = 0
    DefUser#3:
      id = Anon
      name = Anonymus
      lang
      measSystem = 0
    DefUser#4:
      id = Serv
      name = Service
      lang
      measSystem = 0
  Roles:
    DefRole#1:
      id = BR_SecurityAdmin
      level = 100
      admin = TRUE
    DefRole#2:
      id = Administraotr
      level = 100
      admin = TRUE
    DefRole#3:
      id = Operator
      level = 30
      admin = FALSE
    DefRole#4:
      id = Anonymus
      level = 10
      admin = FALSE
    DefRole#5:
      id = Service
      level = 50
      admin = FALSE
```

### Config_1.mpalarmxcore - 5APC3100_KBU1_000/mappServices/Config_1.mpalarmxcore
```
Element gAlarmXCore (Type=mpalarmxcore)
  mapp.Gen:
    Enable = TRUE
    EnableCockpit = FALSE
    EnableOpcUa = FALSE
    TaskClass = 4
    Parent
  mapp.AlarmX.List:
    [0]:
      List = gAlarmXList
      Offset = 0
  mapp.AlarmX.Create = Disabled
  mapp.AlarmX.Core.Retain:
    Memory = 0
```

### Config_1.mpreportcore - 5APC3100_KBU1_000/mappServices/Config_1.mpreportcore
```
Element gReport (Type=mpreportcore)
  mapp.Gen:
    Enable = TRUE
    EnableCockpit = FALSE
    Parent
  MpReport:
    Settings:
      ResourceDeviceName
      LanguageDependent:
        [0]:
          Language = en
          Font = 0
          DateTimePattern = %Y-%m-%d %H:%M:%S
          PrecisionDateTimePattern = %Y-%m-%d %H:%M:%S,%L
        [1]:
          Language = pl
          Font = 0
          DateTimePattern = %Y-%m-%d %H:%M:%S
          PrecisionDateTimePattern = %Y-%m-%d %H:%M:%S,%L
    PageLayouts:
      [0]:
        Name = Default
        PageFormat = 4
        Orientation = 1
        Margins = 1
    Styles:
      Text:
        [0]:
          Name = Default
          Style = 0
          Size = 10
          Color = 000000
          Precision = 6
      Table:
        [0]:
          Name = Default
          BorderWidth = 1
          Color = 000000
          Padding = 1
          HeadRowOnNewPage = FALSE
      Line:
        [0]:
          Name = Default
          Width = 1
          Color = 000000
    Tables:
      [0] = ColumnsByRow
        Name = ResultsTab
        TableStyle = Default
        TextStyle = Default
    Contents:
      [0]:
        Name = ContentHeader
        [0] = Text
          Text = {$IAT/raport_z_gry}
          HorizontalAlign = 0
          NewLine = TRUE
          TextStyle = Default
      [1]:
        Name = ContentLine
        [0] = Line
          LineStyle = Default
      [2]:
        Name = ContentProductionLine
        [0] = Table
          Table = ResultsTab
          HorizontalAlign = 0
    Reports:
      [0]:
        Name = MyReport
        Settings:
          OwnerPassword
          UserPassword
          AllowPrint = TRUE
          AllowCopy = FALSE
          AllowEdit = FALSE
        PageLayout = Default
        Header = ContentHeader
        Footer
        [0]:
          StartOnNewPage = FALSE
          Heading:
            Text
            HorizontalAlign = 0
            TextStyle
          [0]:
            Content = ContentLine
            Width = 100
        [1]:
          StartOnNewPage = FALSE
          Heading:
            Text
            HorizontalAlign = 0
            TextStyle
          [0]:
            Content = ContentProductionLine
            Width = 100
  Alarms = MpAlarmX
    mapp.AlarmX.Core.Configuration:
      [0]:
        Name = GenerateFailed
        Message = {$BR/mapp/MpReportCore/Alarms/GenerateFailed}
        Code = 0
        Severity = 1
        Behavior = EdgeAlarm
          AutoReset = TRUE
          Acknowledge = 1
          Confirm = 0
          MultipleInstances = TRUE
          ReactionWhilePending = TRUE
          Async = FALSE
          Recording:
            InactiveToActive = TRUE
            ActiveToInactive = FALSE
            UnacknowledgedToAcknowledged = TRUE
            UnconfirmedToConfirmed = TRUE
        Disable = FALSE
        AdditionalInformation1
        AdditionalInformation2
```

### Config_2.mpalarmxlist - 5APC3100_KBU1_000/mappServices/Config_2.mpalarmxlist
```
Element gAlarmXList (Type=mpalarmxlist)
  mapp.AlarmX.Core.Configuration:
    [0]:
      Name = MergeError
      Message = Merge się nie powiódł, wołaj Gitmastera
      Code = 0
      Severity = 1
      Behavior = EdgeAlarm
        Confirm = 0
        ReactionWhilePending = TRUE
        Retain = FALSE
        Async = FALSE
        DataUpdate:
          Activation:
            TimeStamp = FALSE
            Snippets = FALSE
        Recording:
          InactiveToActive = TRUE
          UnacknowledgedToAcknowledged = TRUE
          AcknowledgedToUnacknowledged = FALSE
          UnconfirmedToConfirmed = TRUE
          ConfirmedToUnconfirmed = FALSE
      Disable = FALSE
      InhibitPV
      AdditionalInformation1
      AdditionalInformation2
  mapp.AlarmX.Snippets:
    AutoDetect = 1
      Language
```

### Report.mpreportcore - 5APC3100_KBU1_000/mappServices/Report.mpreportcore
```
Element gReport (Type=mpreportcore)
  mapp.Gen:
    Enable = TRUE
    EnableCockpit = FALSE
    Parent
  MpReport:
    Settings:
      ResourceDeviceName = REPORT
      LanguageDependent:
        [0]:
          Language = en
          Font = 0
          DateTimePattern = %Y-%m-%d %H:%M:%S
          PrecisionDateTimePattern = %Y-%m-%d %H:%M:%S,%L
    PageLayouts:
      [0]:
        Name = Layout
        PageFormat = 4
        Orientation = 2
        Margins = 1
    Styles:
      Text:
        [0]:
          Name = Default
          Style = 0
          Size = 10
          Color = 000000
          Precision = 6
    Reports:
      [0]:
        Name
        Settings:
          OwnerPassword
          UserPassword
          AllowPrint = TRUE
          AllowCopy = FALSE
          AllowEdit = FALSE
        PageLayout = Default
        Header
        Footer
        [0]:
          StartOnNewPage = FALSE
          Heading:
            Text
            HorizontalAlign = 0
            TextStyle
  Alarms = MpAlarmX
    mapp.AlarmX.Core.Configuration:
      [0]:
        Name = GenerateFailed
        Message = {$BR/mapp/MpReportCore/Alarms/GenerateFailed}
        Code = 0
        Severity = 1
        Behavior = EdgeAlarm
          AutoReset = TRUE
          Acknowledge = 1
          Confirm = 0
          MultipleInstances = TRUE
          ReactionWhilePending = TRUE
          Async = FALSE
          Recording:
            InactiveToActive = TRUE
            ActiveToInactive = FALSE
            UnacknowledgedToAcknowledged = TRUE
            UnconfirmedToConfirmed = TRUE
        Disable = FALSE
        AdditionalInformation1
        AdditionalInformation2
```

### SaveRecipe.mprecipexml - 5APC3100_KBU1_000/mappServices/SaveRecipe.mprecipexml
```
Element MpLinkgRecipeSR (Type=mprecipexml)
  mapp.Gen:
    Enable = TRUE
    EnableCockpit = FALSE
    TaskClass = 4
    Audit = TRUE
    Parent
  mapp.Recipe.Xml:
    LoadingWarnings = FALSE
    AutoSave = Standard
    Encryption = FALSE
    PassPhrase
    AutoExtension = TRUE
    Signature = Disabled
  Alarms = MpAlarmX
    mapp.AlarmX.Core.Configuration:
      [0]:
        Name = SaveFailed
        Message = {$BR/mapp/MpRecipeXml/Alarms/SaveFailed}
        Code = 0
        Severity = 1
        Behavior = EdgeAlarm
          AutoReset = TRUE
          Acknowledge = 1
          Confirm = 0
          MultipleInstances = TRUE
          ReactionWhilePending = TRUE
          Async = FALSE
          Recording:
            InactiveToActive = TRUE
            ActiveToInactive = FALSE
            UnacknowledgedToAcknowledged = TRUE
            UnconfirmedToConfirmed = TRUE
        Disable = FALSE
        AdditionalInformation1
        AdditionalInformation2
      [1]:
        Name = SaveFailedPartial
        Message = {$BR/mapp/MpRecipeXml/Alarms/SaveFailedPartial}
        Code = 0
        Severity = 1
        Behavior = EdgeAlarm
          AutoReset = TRUE
          Acknowledge = 1
          Confirm = 0
          MultipleInstances = TRUE
          ReactionWhilePending = TRUE
          Async = FALSE
          Recording:
            InactiveToActive = TRUE
            ActiveToInactive = FALSE
            UnacknowledgedToAcknowledged = TRUE
            UnconfirmedToConfirmed = TRUE
        Disable = FALSE
        AdditionalInformation1
        AdditionalInformation2
      [2]:
        Name = LoadFailed
        Message = {$BR/mapp/MpRecipeXml/Alarms/LoadFailed}
        Code = 0
        Severity = 1
        Behavior = EdgeAlarm
          AutoReset = TRUE
          Acknowledge = 1
          Confirm = 0
          MultipleInstances = TRUE
          ReactionWhilePending = TRUE
          Async = FALSE
          Recording:
            InactiveToActive = TRUE
            ActiveToInactive = FALSE
            UnacknowledgedToAcknowledged = TRUE
            UnconfirmedToConfirmed = TRUE
        Disable = FALSE
        AdditionalInformation1
        AdditionalInformation2
      [3]:
        Name = LoadFailedPartial
        Message = {$BR/mapp/MpRecipeXml/Alarms/LoadFailedPartial}
        Code = 0
        Severity = 1
        Behavior = EdgeAlarm
          AutoReset = TRUE
          Acknowledge = 1
          Confirm = 0
          MultipleInstances = TRUE
          ReactionWhilePending = TRUE
          Async = FALSE
          Recording:
            InactiveToActive = TRUE
            ActiveToInactive = FALSE
            UnacknowledgedToAcknowledged = TRUE
            UnconfirmedToConfirmed = TRUE
        Disable = FALSE
        AdditionalInformation1
        AdditionalInformation2
```

### Settings.vicfg - 5APC3100_KBU1_000/mappVision/Settings.vicfg
```
Element VisionSettings (Type=vicfg)
  ActivateVisualization = TRUE
  FileDeviceName
  Protocol = Unsecure
  DeepLearning:
    CustomDlNetworks:
      DLFileDeviceName
      DLNetworkBuildPath
```

### viComp.visioncomponent - 5APC3100_KBU1_000/mappVision/viComp.visioncomponent
```
Element gCamera (Type=visioncomponent)
  VisionApplicationReference = ViApplication
  CalibrationSelections
```

## Logical view

Binary libraries used (declarations not repeated): operator, runtime, AsIecCon, McBase, McAcpAx, MpRobotics 6.7.2, McAxGroup, McPathGen, MpAxis, CoTrace, McAxis, McAcpPar 6.7.2, FileIO, sys_lib, AsBrStr, MpBase, McProgInt, astime, ViBase 6.7.0, AsZip, AsARCfg, powerlnk, AsEPL, AsIO, AsTCP, DataObj, ArSsl, MpAlarmX, MpServer, MpRecipe, MpFile, MpAudit 6.7.1, MpReport 6.7.1, standard

### Global.typ - Global data types
```iecst
TYPE
	AlarmEnum : 	STRUCT
		EstopActive : BOOL; (*E stop zostal zalaczony*)
		InncorrectRobotMove : BOOL; (*Zle przeniesienie pionka przez robota*)
		InncorrectBoard : BOOL; (*Zla plansza do startu gry*)
		FolderError : USINT; (*blad folderu*)
		MissingSTMotionProgram : USINT; (*Brakuje programu ST Motion*)
		RobotProgramNotLoaded : BOOL; (*Program (napisany w STMotion) nie istnieje w pamiďż˝ci USER robota*)
		RobotWorkspaceViolation : BOOL; (*TCP robota znalazďż˝o siďż˝ poza dozwolonym obszarem - robot nie moďż˝e kontynuowaďż˝ ruchu w tym kierunku*)
		RobotAxisViolation : BOOL; (*Robota przekroczyďż˝ maksymalnďż˝ pozycjďż˝ kďż˝towďż˝ w ktďż˝rejďż˝ z osi*)
		RobotRestorePosFail : BOOL; (*Nie udało się wykonać bazowania za pomocą restore pos podczas uruchamiania robota*)
	END_STRUCT;
	GameEnum : 	STRUCT
		BoardActual : ARRAY[1..8,1..8]OF USINT;
		gPickPiece : ARRAY[1..8,1..8]OF BOOL;
		gEnableMove : ARRAY[1..8,1..8]OF BOOL;
		gPickMove : ARRAY[1..8,1..8]OF BOOL;
		gEnablePiece : ARRAY[1..8,1..8]OF BOOL;
	END_STRUCT;
	GameStatStruct : 	STRUCT
		MoveCount : INT;
		MoveHistory : ARRAY[1..4]OF STRING[20];
		Load : BOOL;
	END_STRUCT;
	StepEnum :
		(
		Idle, (*Czekanie na start = 1*)
		PhotoCheck, (*Drugie zdjecie sprawdzajace poprawnosci odlozenia pionkow po ruchu*)
		GameMove, (*Ruch warcabowy człowiek vs AI*)
		RobotMove, (*Robot wykonuje fizyczny ruch*)
		ErrorState,
		ResetRobotPos,
		SetBoard,
		SetBoardPrep
		);
END_TYPE
```

### Global.var - Global variables
```iecst
VAR
	gCameraEnd : BOOL;
	gBoardCamera : ARRAY[1..8,1..8] OF USINT;
	gAlarm : AlarmEnum;
	gGame : USINT;
	gPickPiece : ARRAY[1..8,1..8] OF BOOL; (*Klikniety przez gracza pionek*)
	gEnableMove : ARRAY[1..8,1..8] OF BOOL; (*Mozliwe ruchy na szachownicy*)
	gPickMove : ARRAY[1..8,1..8] OF BOOL; (*Wybrany ruch przez gracza*)
	gBoardActual : ARRAY[1..8,1..8] OF USINT; (*Aktualna plansza rozgrywki (0 puste pole, 1 biale, 2 czarne, 3 damka biale, 4 damka czarne)*)
	gGameRound : BOOL; (*False ruch robota, True ruch czlowieka*)
	gPlayerColor : BOOL; (*True - biale, False - czarne*)
	gDifficultyLevel : USINT; (*0 - Easy, 1 - Medium, 2 - Hard*)
	gStart : BOOL; (*True - rozpocznij nowa gre, False - nic*)
	gEnablePiece : ARRAY[1..8,1..8] OF BOOL; (*Pionki mozliwe do klikniecia podczas tury*)
	gESTOP : BOOL; (*Sygnal z sterownika Safety*)
	gStep : StepEnum; (*Maszyna stanow robota*)
	gGameStats : GameStatStruct; (*Statystyki gry*)
	gCameraEnd : BOOL;
	gCameraTrigger : BOOL;
	gBoardCamera : ARRAY[1..8,1..8] OF USINT;
END_VAR
```

### Package Logical/Libraries - Global libraries

### Library Logical/Libraries/CameraMath (IEC)

#### CameraMath.fun - Exported functions and function blocks
```iecst
FUNCTION CalculateTransformation : BOOL

	VAR_INPUT

		ReferenceMarker3X : DINT;
		ReferenceMarker3Y : DINT;

		ReferenceMarker4X : DINT;
		ReferenceMarker4Y : DINT;

		CurrentMarker3X : DINT;
		CurrentMarker3Y : DINT;

		CurrentMarker4X : DINT;
		CurrentMarker4Y : DINT;

	END_VAR

	VAR_IN_OUT

		TransformationA : LREAL;
		TransformationB : LREAL;
		TransformationDen : LREAL;

	END_VAR

	VAR

		referenceVectorX : LREAL;
		referenceVectorY : LREAL;

		currentVectorX : LREAL;
		currentVectorY : LREAL;

		referenceDen : LREAL;

	END_VAR

END_FUNCTION
```

#### CalculateTransformation.st - not listed in the package file held
```iecst
FUNCTION CalculateTransformation

	referenceVectorX := DINT_TO_LREAL(ReferenceMarker4X - ReferenceMarker3X);

	referenceVectorY := DINT_TO_LREAL(ReferenceMarker4Y - ReferenceMarker3Y);

	currentVectorX := DINT_TO_LREAL(CurrentMarker4X - CurrentMarker3X);

	currentVectorY := DINT_TO_LREAL(CurrentMarker4Y - CurrentMarker3Y);

	referenceDen := (referenceVectorX * referenceVectorX) + (referenceVectorY * referenceVectorY);

	IF referenceDen > 0.0 THEN

		TransformationA := ((currentVectorX * referenceVectorX) + (currentVectorY * referenceVectorY)) / referenceDen;

		TransformationB := ((currentVectorY * referenceVectorX) - (currentVectorX * referenceVectorY)) / referenceDen;

		TransformationDen := (TransformationA * TransformationA) + (TransformationB * TransformationB);

		CalculateTransformation := TransformationDen > 0.0;

	ELSE

		TransformationA := 0.0;
		TransformationB := 0.0;
		TransformationDen := 0.0;
		CalculateTransformation := FALSE;
	END_IF;

END_FUNCTION
```

- Visualisation Logical/mappView (not shown)

### MotionInterface.typ
```iecst
TYPE
	JogCartesianType : 	STRUCT
		JogXPos : BOOL;
		JogXNeg : BOOL;
		JogYPos : BOOL;
		JogYNeg : BOOL;
		JogZPos : BOOL;
		JogZNeg : BOOL;
		Speed : REAL := 30;
	END_STRUCT;
	JogJointType : 	STRUCT
		JogPos0 : BOOL;
		JogPos1 : BOOL;
		JogPos2 : BOOL;
		JogPos3 : BOOL;
		JogPos4 : BOOL;
		JogPos5 : BOOL;
		JogNeg0 : BOOL;
		JogNeg1 : BOOL;
		JogNeg2 : BOOL;
		JogNeg3 : BOOL;
		JogNeg4 : BOOL;
		JogNeg5 : BOOL;
		Speed : REAL := 30;
	END_STRUCT;
	ManualType : 	STRUCT
		Joint : JogJointType;
		Cartesian : JogCartesianType;
		RequestRehomeRobot : BOOL;
		RequestGoHome : BOOL;
		UsingUCS : BOOL;
	END_STRUCT;
	MotionInterfaceType : 	STRUCT
		RequestManualMode : BOOL;
		StartPos : McPosType; (*Skąd przenieść pionek*)
		EndPos : McPosType;
		WhitePilePos : McPosType; (*Pozycja 1szego miejsca na stosie, reszta jest juz obliczana przez program*)
		BlackPilePos : McPosType; (*Pozycja 1szego miejsca na stosie, reszta jest juz obliczana przez program*)
		Feedrate : RobotFeedrateType;
		Command : RobotCommandType; (*Przesunięcie warcaba ze StartPos na EndPos*)
		Ready : BOOL;
		ReadyToPowerOn : BOOL;
		Execute : BOOL; (*Najlepiej podac impuls*)
		Busy : BOOL;
		Done : BOOL;
		Manual : ManualType;
		Enable : BOOL;
	END_STRUCT;
	RobotCommandType :
		(
		MOVE_HOME,
		DISCARD_WHITE,
		DISCARD_BLACK,
		MOVE_START_END (*Przesuniecie ze StartPos na EndPos*)
		);
	RobotMoveVarType : 	STRUCT
		DiscardColor : USINT := 0;
		Capture : BOOL := FALSE;
		StartPoint : IndexPointType;
		EndPoint : IndexPointType;
		DiscardPoint : IndexPointType;
		RTRMove : BOOL := FALSE; (*Ready to read move*)
	END_STRUCT;
	IndexPointType : 	STRUCT
		x : USINT := 1;
		y : USINT := 1;
	END_STRUCT;
	RobotFeedrateType : 	STRUCT
		High : LREAL := 10000;
		Low : LREAL := 1500;
	END_STRUCT;
END_TYPE
```

### MotionInterface.var
```iecst
VAR
	gRobotMoveVar : RobotMoveVarType;
	gMotionInterface : MotionInterfaceType;
END_VAR
```

### Robot.var - Local variables
```iecst
VAR
	Robot : MpRoboArm6Axis;
	RobotPar : MpRoboArm6AxisParType;
	doMagnet : BOOL;
	WorkspaceMonitor : McPathGenMonElemWorkspaceType;
END_VAR
VAR RETAIN
	AxisRestorePos0 : {REDUND_UNREPLICABLE} McAcpAxRestorePosType;
	AxisRestorePos1 : {REDUND_UNREPLICABLE} McAcpAxRestorePosType;
	AxisRestorePos2 : {REDUND_UNREPLICABLE} McAcpAxRestorePosType;
	AxisRestorePos3 : {REDUND_UNREPLICABLE} McAcpAxRestorePosType;
	AxisRestorePos4 : {REDUND_UNREPLICABLE} McAcpAxRestorePosType;
	AxisRestorePos5 : {REDUND_UNREPLICABLE} McAcpAxRestorePosType;
	RestorePosReady : BOOL;
END_VAR
```

### Program Logical/Programs/Motion/MotionCtrl (IEC)

#### Main.st - Init, cyclic, exit code
```iecst
PROGRAM _INIT
	doMagnet;

	gESTOP := TRUE;

	gAxesGroup_Racer3_1;
	gAxisQ1_Racer3_1;
	gAxisQ2_Racer3_1;
	gAxisQ3_Racer3_1;
	gAxisQ4_Racer3_1;
	gAxisQ5_Racer3_1;
	gAxisQ6_Racer3_1;

	STMotionHomePoint;

	mcGroupHome.AxesGroup := ADR(gAxesGroup_Racer3_1);

	Robot.MpLink := ADR(gAxesGroup_Racer3_1);
	Robot.Enable := 1;
	Robot.ErrorReset := 0;
	Robot.Parameters := ADR(RobotPar);
	Robot.Update := 1;
	Robot.Override := 100;
	Robot.Power := 0;
	Robot();

	RobotState := ROBOT_ENABLED;

	PauseWorkspaceMonitoring.AxesGroup := ADR(gAxesGroup_Racer3_1);
	PauseWorkspaceMonitoring.Enable := FALSE;

END_PROGRAM

PROGRAM _CYCLIC
	// TRZEBA ZROBIĆ SYNCHRONIZACJE
	ExecuteImpulse := RTrigExecute.Q;
	RTrigExecute.CLK := gMotionInterface.Execute;

	STMotionDoneImpulse := RTrigSTMotionDone.Q;
	RTrigSTMotionDone.CLK := STMotionDone;

	gMotionInterface.Ready := FALSE;
	gMotionInterface.ReadyToPowerOn := FALSE;

	CASE RobotState OF
		ROBOT_DISABLED:
			gMotionInterface.ReadyToPowerOn := TRUE;
			IF gMotionInterface.Enable THEN
				RobotState := ROBOT_ENABLED;
				Robot.ErrorReset := 0;
			END_IF;

		ROBOT_ENABLED:
			Robot.Power := TRUE;
			IF Robot.PowerOn THEN
				RobotState := ROBOT_HOMING_SELECT;
			END_IF;

		ROBOT_HOMING_SELECT:
			// Bazowanie Restore Position
			IF RestorePosReady THEN
				RobotState := ROBOT_HOMING_RESTORE;
			// Bazowanie Homing Direct
			ELSE
				RobotState := ROBOT_HOMING_DIRECT;
			END_IF;

		ROBOT_HOMING_DIRECT:
			FOR i := 0 TO 5 DO
				mcGroupHome.HomingMode[i] := mcHOMING_DIRECT;
				mcGroupHome.Position[i] := AxisPos[i];
			END_FOR;
			mcGroupHome.Execute := TRUE;
			IF mcGroupHome.Done THEN
				RobotState := ROBOT_HOMED;
				gMotionInterface.Manual.RequestRehomeRobot := FALSE;
				RestorePosReady := TRUE;
				mcGroupHome.Execute := FALSE;
			END_IF;

		ROBOT_HOMING_RESTORE:
			FOR i := 0 TO 5 DO
				mcGroupHome.HomingMode[i] := mcHOMING_RESTORE_POSITION;
				mcGroupHome.Position[i] := AxisPos[i];
			END_FOR;
			mcGroupHome.Execute := TRUE;
			IF mcGroupHome.Done THEN
				RobotState := ROBOT_HOMED;
				mcGroupHome.Execute := FALSE;
			END_IF;

		ROBOT_HOMED:

			gMotionInterface.Ready := TRUE;

			gMotionInterface.Done := FALSE;
			IF gMotionInterface.RequestManualMode THEN
				RobotState := ROBOT_MANUAL;
			ELSIF ExecuteImpulse  THEN
				RobotState := ROBOT_EXECUTE;
			END_IF;

		ROBOT_MANUAL:
			// domyslnie

			RobotPar.Jog.Velocity[0] := 0;
			RobotPar.Jog.Velocity[1] := 0;
			RobotPar.Jog.Velocity[2] := 0;
			RobotPar.Jog.Velocity[3] := 0;
			RobotPar.Jog.Velocity[4] := 0;
			RobotPar.Jog.Velocity[5] := 0;
			Robot.Jog := FALSE;

			JogJointPos0 := gMotionInterface.Manual.Joint.JogPos0;
			JogJointPos1 := gMotionInterface.Manual.Joint.JogPos1;
			JogJointPos2 := gMotionInterface.Manual.Joint.JogPos2;
			JogJointPos3 := gMotionInterface.Manual.Joint.JogPos3;
			JogJointPos4 := gMotionInterface.Manual.Joint.JogPos4;
			JogJointPos5 := gMotionInterface.Manual.Joint.JogPos5;
			JogJointNeg0 := gMotionInterface.Manual.Joint.JogNeg0;
			JogJointNeg1 := gMotionInterface.Manual.Joint.JogNeg1;
			JogJointNeg2 := gMotionInterface.Manual.Joint.JogNeg2;
			JogJointNeg3 := gMotionInterface.Manual.Joint.JogNeg3;
			JogJointNeg4 := gMotionInterface.Manual.Joint.JogNeg4;
			JogJointNeg5 := gMotionInterface.Manual.Joint.JogNeg5;
			JogJointSpeed := gMotionInterface.Manual.Joint.Speed;

			JogXPos := gMotionInterface.Manual.Cartesian.JogXPos;
			JogXNeg := gMotionInterface.Manual.Cartesian.JogXNeg;
			JogYPos := gMotionInterface.Manual.Cartesian.JogYPos;
			JogYNeg := gMotionInterface.Manual.Cartesian.JogYNeg;
			JogZPos := gMotionInterface.Manual.Cartesian.JogZPos;
			JogZNeg := gMotionInterface.Manual.Cartesian.JogZNeg;
			JogCartesianSpeed := gMotionInterface.Manual.Cartesian.Speed;

			JogJointAny := JogJointPos0 OR JogJointNeg0
			OR JogJointPos1 OR JogJointNeg1
			OR JogJointPos2 OR JogJointNeg2
			OR JogJointPos3 OR JogJointNeg3
			OR JogJointPos4 OR JogJointNeg4
			OR JogJointPos5 OR JogJointNeg5;

			IF JogJointAny THEN
				// tryb JogJoint
				RobotPar.Jog.CoordSystem := mcJACS;

				IF JogJointPos0 THEN
					RobotPar.Jog.Velocity[0] := JogJointSpeed;
				ELSIF JogJointNeg0 THEN
					RobotPar.Jog.Velocity[0] := -JogJointSpeed;
				END_IF;
				IF JogJointPos1 THEN
					RobotPar.Jog.Velocity[1] := JogJointSpeed;
				ELSIF JogJointNeg1 THEN
					RobotPar.Jog.Velocity[1] := -JogJointSpeed;
				END_IF;
				IF JogJointPos2 THEN
					RobotPar.Jog.Velocity[2] := JogJointSpeed;
				ELSIF JogJointNeg2 THEN
					RobotPar.Jog.Velocity[2] := -JogJointSpeed;
				END_IF;
				IF JogJointPos3 THEN
					RobotPar.Jog.Velocity[3] := JogJointSpeed;
				ELSIF JogJointNeg3 THEN
					RobotPar.Jog.Velocity[3] := -JogJointSpeed;
				END_IF;
				IF JogJointPos4 THEN
					RobotPar.Jog.Velocity[4] := JogJointSpeed;
				ELSIF JogJointNeg4 THEN
					RobotPar.Jog.Velocity[4] := -JogJointSpeed;
				END_IF;
				IF JogJointPos5 THEN
					RobotPar.Jog.Velocity[5] := JogJointSpeed;
				ELSIF JogJointNeg5 THEN
					RobotPar.Jog.Velocity[5] := -JogJointSpeed;
				END_IF;

				Robot.Jog := TRUE;
			ELSIF JogXPos OR JogXNeg OR JogYPos OR JogYNeg OR JogZPos OR JogZNeg THEN
				// tryb JogCartesian
				RobotPar.Jog.CoordSystem := mcMCS; // lub inny
				Robot.Jog := TRUE;

				IF JogXPos THEN
					RobotPar.Jog.Velocity[0] := JogCartesianSpeed;
				END_IF;
				IF JogXNeg THEN
					RobotPar.Jog.Velocity[0] := -JogCartesianSpeed;
					END_IF;
				IF JogYPos THEN
					RobotPar.Jog.Velocity[1] := JogCartesianSpeed;
				END_IF;
				IF JogYNeg THEN
					RobotPar.Jog.Velocity[1] := -JogCartesianSpeed;
				END_IF;
				IF JogZPos THEN
					RobotPar.Jog.Velocity[2] := JogCartesianSpeed;
				END_IF;
				IF JogZNeg THEN
					RobotPar.Jog.Velocity[2] := -JogCartesianSpeed;
				END_IF;

			ELSIF gMotionInterface.Manual.RequestGoHome THEN
				RobotPar.ProgramName := 'gohome.st';
				Robot.MoveProgram := TRUE;
				STMotionDone := FALSE;
				STMotionLowFeedrate := gMotionInterface.Feedrate.Low;
				PauseWorkspaceMonitoring.Enable := TRUE;
				RobotState := ROBOT_GO_HOME;
				gMotionInterface.Manual.RequestGoHome := FALSE;
			END_IF;

			IF NOT gMotionInterface.RequestManualMode THEN
				gAlarm.RobotRestorePosFail := FALSE;
				Robot.Jog := FALSE;
				RobotState := ROBOT_HOMED;
			END_IF;

			IF gMotionInterface.Manual.RequestRehomeRobot THEN
				gAlarm.RobotRestorePosFail := FALSE;
				gMotionInterface.Manual.RequestRehomeRobot := FALSE;

				Robot.Jog := FALSE;
				RobotState := ROBOT_HOMING_DIRECT;
			END_IF;

			IF STMotionDoneImpulse THEN
				Robot.MoveProgram := FALSE;
				Robot.Interrupt := TRUE;
			END_IF;

		ROBOT_GO_HOME:
			IF STMotionDone THEN
				PauseWorkspaceMonitoring.Enable := FALSE;
				RobotState := ROBOT_MANUAL;
			END_IF;

		ROBOT_EXECUTE:

			STMotionHighFeedrate := gMotionInterface.Feedrate.High;
			STMotionLowFeedrate := gMotionInterface.Feedrate.Low;

			// Ustalanie na jaka pozycje warcab ma byc odstawiony
			CASE gMotionInterface.Command OF
				MOVE_START_END:
					STMotionStartPoint.Pos := gMotionInterface.StartPos;
					STMotionStartPoint.Orient := STMotionDefaultOrient;
					STMotionEndPoint.Pos := gMotionInterface.EndPos;
					STMotionEndPoint.Orient := STMotionDefaultOrient;
					RobotPar.ProgramName := 'moveAB.st';
				MOVE_HOME:
					RobotPar.ProgramName := 'move.st';
				DISCARD_WHITE:
					PileCalculatedOffs.X := WhitePileXOffs * USINT_TO_REAL(WhitePileCnt/PileHeight);
					PileCalculatedOffs.Y := WhitePileYOffs * USINT_TO_REAL(WhitePileCnt MOD PileHeight);
					PileCalculatedOffs.Z := 0;

					STMotionEndPoint.Pos.X := gMotionInterface.WhitePilePos.X + PileCalculatedOffs.X;
					STMotionEndPoint.Pos.Y := gMotionInterface.WhitePilePos.Y + PileCalculatedOffs.Y;
					STMotionEndPoint.Pos.Z := gMotionInterface.WhitePilePos.Z + PileCalculatedOffs.Z;
					STMotionEndPoint.Orient := STMotionDefaultOrient;
					RobotPar.ProgramName := 'moveAB.st';
				DISCARD_BLACK:
					PileCalculatedOffs.X := BlackPileXOffs * USINT_TO_REAL(BlackPileCnt/PileHeight);
					PileCalculatedOffs.Y := BlackPileYOffs * USINT_TO_REAL(BlackPileCnt MOD PileHeight);
					PileCalculatedOffs.Z := 0;

					STMotionEndPoint.Pos.X := gMotionInterface.BlackPilePos.X + PileCalculatedOffs.X;
					STMotionEndPoint.Pos.Y := gMotionInterface.BlackPilePos.Y + PileCalculatedOffs.Y;
					STMotionEndPoint.Pos.Z := gMotionInterface.BlackPilePos.Z + PileCalculatedOffs.Z;
					STMotionEndPoint.Orient := STMotionDefaultOrient;
					RobotPar.ProgramName := 'moveAB.st';
			END_CASE;

			// rozpoczecie pracy programu

			Robot.Interrupt := FALSE;
			Robot.MoveProgram := TRUE;

			STMotionDone := FALSE;
			gMotionInterface.Busy := TRUE;
			RobotState := ROBOT_MOVING;

		ROBOT_MOVING:
			IF STMotionDone THEN
				gMotionInterface.Busy := FALSE;
				Robot.MoveProgram := FALSE;
				STMotionDone := FALSE;
				gMotionInterface.Done := TRUE;
				RobotState := ROBOT_MOVE_DONE;
				Robot.Interrupt := TRUE;
			END_IF;

		ROBOT_MOVE_DONE:
			IF NOT gMotionInterface.Execute THEN
				gMotionInterface.Done := FALSE;
				Robot.Interrupt := FALSE;
				RobotState := ROBOT_HOMED;
			END_IF;

	END_CASE;

	IF NOT (RobotState = ROBOT_MANUAL OR RobotState = ROBOT_MOVING) THEN
		doMagnet := FALSE;
	END_IF;

	IF NOT gMotionInterface.Enable THEN
		gMotionInterface.Busy := 0;
		RobotState := ROBOT_DISABLED;
		gMotionInterface.Execute := 0;
		Robot.ErrorReset := 1;
		Robot.Power := 0;
		mcGroupHome.Execute := 0;
		Robot.Jog := 0;
		Robot.MoveProgram := 0;
		Robot.Interrupt := 1;
	END_IF;

	gESTOP := Robot.Info.ReadyToPowerOn;

	PauseWorkspaceMonitoring();
	RTrigSTMotionDone();
	RTrigExecute();
	mcGroupHome();
	Robot();
END_PROGRAM

PROGRAM _EXIT

END_PROGRAM
```

#### Types.typ - Local data types
```iecst
TYPE
	RobotStateType :
		(
		ROBOT_DISABLED,
		ROBOT_ENABLED,
		ROBOT_HOMING_SELECT,
		ROBOT_HOMING_DIRECT,
		ROBOT_HOMING_RESTORE,
		ROBOT_HOMED,
		ROBOT_MANUAL,
		ROBOT_GO_HOME,
		ROBOT_EXECUTE,
		ROBOT_MOVING,
		ROBOT_MOVE_DONE
		);
END_TYPE
```

#### Variables.var
```iecst
(* Sterowanie robotem i homing *)
VAR
	RobotState : RobotStateType := ROBOT_DISABLED;
	mcGroupHome : MC_BR_GroupHome_15;
	AxisPos : ARRAY[0..5] OF REAL := [2(0),-90,3(0)];
	i : USINT;
	PauseWorkspaceMonitoring : MC_BR_PauseWorkspaceMonitoring;
END_VAR
(* Wymiana danych z ST Motion *)
VAR
	STMotionStartPoint : McPointType;
	STMotionEndPoint : McPointType;
	STMotionHomePoint : McPointType := (Pos:=(X:=290,Y:=-205,Z:=494),Orient:=(Angle1:=0,Angle2:=180,Angle3:=0));
	STMotionDone : BOOL := FALSE;
END_VAR
VAR CONSTANT
	STMotionDefaultOrient : McOrientType := (Angle1:=0,Angle2:=180,Angle3:=0);
END_VAR
VAR
	STMotionHighFeedrate : LREAL := 5000;
	STMotionLowFeedrate : LREAL := 500;
END_VAR
(* Synchronizacja PLC ze ST Motion *)
VAR
	RTrigExecute : r_trig;
	ExecuteImpulse : BOOL;
	RTrigSTMotionDone : r_trig;
	STMotionDoneImpulse : BOOL;
END_VAR
(* Obs³uga stosów warcabów *)
VAR CONSTANT
	BlackPileXOffs : REAL := 50;
	WhitePileXOffs : REAL := -50;
	BlackPileYOffs : REAL := 0.0;
	WhitePileYOffs : REAL := 0.0;
	PileZOffs : REAL := 0;
	PileHeight : USINT := 4;
END_VAR
VAR
	BlackPileCnt : USINT;
	WhitePileCnt : USINT;
	PileCalculatedOffs : McPosType;
END_VAR
(* Rêczne sterowanie kartezjañskie *)
VAR
	JogXPos : BOOL;
	JogXNeg : BOOL;
	JogYPos : BOOL;
	JogYNeg : BOOL;
	JogZPos : BOOL;
	JogZNeg : BOOL;
	JogCartesianSpeed : REAL;
END_VAR
(* Rêczne sterowanie osiami robota *)
VAR
	JogJointPos0 : BOOL;
	JogJointNeg0 : BOOL;
	JogJointPos1 : BOOL;
	JogJointNeg1 : BOOL;
	JogJointPos2 : BOOL;
	JogJointNeg2 : BOOL;
	JogJointPos3 : BOOL;
	JogJointNeg3 : BOOL;
	JogJointPos4 : BOOL;
	JogJointNeg4 : BOOL;
	JogJointPos5 : BOOL;
	JogJointNeg5 : BOOL;
	JogJointAny : BOOL;
	JogJointSpeed : REAL;
END_VAR
```

#### Types1.typ - not listed in the package file held
```iecst
TYPE
	RobotStateType :
		(
		ROBOT_DISABLED,
		ROBOT_ENABLED,
		ROBOT_POWERED,
		ROBOT_HOMED,
		ROBOT_MANUAL,
		ROBOT_EXECUTE
		);
END_TYPE
```

### Program Logical/Programs/Motion/PositionInfo (IEC)

#### Variables.var
```iecst
VAR
	AxisQ1Pos : LREAL;
	AxisQ2Pos : LREAL;
	AxisQ3Pos : LREAL;
	AxisQ4Pos : LREAL;
	AxisQ5Pos : LREAL;
	AxisQ6Pos : LREAL;
	X : LREAL;
	Y : LREAL;
	Z : LREAL;
	GetCoordSystemIdent : MC_BR_GetCoordSystemIdent;
	ReadActualPosition : MC_GroupReadActualPosition_15;
END_VAR
```

#### Main.st
```iecst
PROGRAM _INIT
	AxisRestorePos0;
	AxisRestorePos1;
	AxisRestorePos2;
	AxisRestorePos3;
	AxisRestorePos4;
	AxisRestorePos5;

	GetCoordSystemIdent.Execute := TRUE;
	GetCoordSystemIdent.CoordSystemName := 'gUserFrame';

	GetCoordSystemIdent();

	ReadActualPosition.AxesGroup := ADR(gAxesGroup_Racer3_1);
	ReadActualPosition.Enable := TRUE;
	ReadActualPosition.CoordSystem := GetCoordSystemIdent.Ident;
END_PROGRAM

PROGRAM _CYCLIC

	AxisQ1Pos := -Robot.Info.JointAxisPosition[0];
	AxisQ2Pos := Robot.Info.JointAxisPosition[1];
	AxisQ3Pos := -Robot.Info.JointAxisPosition[2];
	AxisQ4Pos := -Robot.Info.JointAxisPosition[3];
	AxisQ5Pos := Robot.Info.JointAxisPosition[4];
	AxisQ6Pos := -Robot.Info.JointAxisPosition[5];

	IF gMotionInterface.Manual.UsingUCS THEN

		X := ReadActualPosition.Position[0];
		Y := ReadActualPosition.Position[1];
		Z := ReadActualPosition.Position[2];
	ELSE
		X := Robot.X;
		Y := Robot.Y;
		Z := Robot.Z;
	END_IF;

	gAlarm.RobotWorkspaceViolation := 0;
	gAlarm.RobotAxisViolation := 0;

	IF WorkspaceMonitor.WorkspaceStatus = mcPATHGEN_WS_WORKSPACE_VIOLATION
		OR WorkspaceMonitor.WorkspaceStatus = mcPATHGEN_WS_SAFESPACE_VIOLATION
		OR WorkspaceMonitor.WorkspaceStatus = mcPATHGEN_WS_WORKRANGE_VIOLATION THEN
		gAlarm.RobotWorkspaceViolation := 1;
	END_IF;
	IF WorkspaceMonitor.WorkspaceStatus = mcPATHGEN_WS_AXES_VIOLATION
		OR WorkspaceMonitor.WorkspaceStatus = mcPATHGEN_WS_JOINTAXES_VIOLATION THEN
		gAlarm.RobotAxisViolation := 1;
	END_IF;

	IF NOT RestorePosReady THEN
		gAlarm.RobotRestorePosFail := TRUE;
	ELSE
		gAlarm.RobotRestorePosFail := FALSE;
	END_IF;

	GetCoordSystemIdent();
	ReadActualPosition();

END_PROGRAM

PROGRAM _EXIT

END_PROGRAM
```

### Types.typ - not listed in the package file held
```iecst
TYPE
	RobotStateType :
		(
		ROBOT_DISABLED,
		ROBOT_ENABLED,
		ROBOT_POWERED,
		ROBOT_HOMED,
		ROBOT_MANUAL
		);
END_TYPE
```

### Variables.var - not listed in the package file held
```iecst
VAR
	Robot : MpRoboArm6Axis;
	RobotPar : MpRoboArm6AxisParType;
	mcGroupHome : MC_BR_GroupHome_15;
END_VAR
(*Jog Joint*)
VAR
	SelJoint : USINT; (*Stawy sa liczone od 0 do 5*)
	JogJointPos : BOOL;
	JogJointNeg : BOOL;
END_VAR
(*Jog Cartesian*)
VAR
	JogXPos : BOOL;
	JogXNeg : BOOL;
	JogYPos : BOOL;
	JogYNeg : BOOL;
	JogZPos : BOOL;
	JogZNeg : BOOL;
END_VAR
(*Jog Param*)
VAR
	JogJointSpeed : REAL := 20;
	JogCartesianSpeed : REAL := 20;
END_VAR
(*Parametry Home*)
VAR
	AxisPos : ARRAY[0..5] OF REAL := [2(0),-90,0,90,0];
	RobotState : RobotStateType;
END_VAR
```

### Program Logical/Programs/Motion/FixAxisDir

#### Variables.var
```iecst
VAR
	AxisQ1Pos : LREAL;
	AxisQ2Pos : LREAL;
	AxisQ3Pos : LREAL;
	AxisQ4Pos : LREAL;
	AxisQ5Pos : LREAL;
	AxisQ6Pos : LREAL;
END_VAR
```

#### Main.st
```iecst
PROGRAM _INIT

END_PROGRAM

PROGRAM _CYCLIC
	AxisQ1Pos := -Robot.Info.JointAxisPosition[0];
	AxisQ2Pos := Robot.Info.JointAxisPosition[1];
	AxisQ3Pos := -Robot.Info.JointAxisPosition[2];
	AxisQ4Pos := Robot.Info.JointAxisPosition[3];
	AxisQ5Pos := Robot.Info.JointAxisPosition[4];
	AxisQ6Pos := Robot.Info.JointAxisPosition[5];
END_PROGRAM

PROGRAM _EXIT

END_PROGRAM
```

### Program Logical/Programs/Motion/Program

#### Variables.var
```iecst
VAR
	Robot : MpRoboArm6Axis;
	RobotPar : MpRoboArm6AxisParType;
END_VAR
```

#### Main.st
```iecst
PROGRAM _INIT
	(* Insert code here *)
	gAxesGroup_Racer3_1;
	gAxisQ1_Racer3_1;
	gAxisQ2_Racer3_1;
	gAxisQ3_Racer3_1;
	gAxisQ4_Racer3_1;
	gAxisQ5_Racer3_1;
	gAxisQ6_Racer3_1;

	Robot.MpLink := ADR(gAxesGroup_Racer3_1);
	Robot.Enable := 1;
	Robot.ErrorReset := 0;
	Robot.Parameters := ADR(RobotPar);
	Robot.Update := 1;
	Robot();

END_PROGRAM

PROGRAM _CYCLIC
	(* Insert code here *)
	Robot.Update := 0;
	Robot();

END_PROGRAM

PROGRAM _EXIT
	(* Insert code here *)

END_PROGRAM
```

### Program Logical/Programs/Motion/RobotMove

#### Types.typ
```iecst
TYPE
	RobotMoveEnum :
		(
		IdleRM,
		MoveExecute,
		MoveBusy,
		DiscardExecute,
		DiscardBusy,
		EndRM
		);
END_TYPE
```

#### Variables.var
```iecst
VAR
	MoveStep : RobotMoveEnum := Idle;
	Doing : BOOL;
	COORD_POSITION : ARRAY[1..8,1..8] OF McPosType := [
	(X:=546.0, Y:=-122.0, Z:=221.2), (X:=504.1, Y:=-121.8, Z:=221.2), (X:=462.1, Y:=-121.7, Z:=221.3), (X:=420.2, Y:=-121.5, Z:=221.3),
	(X:=378.2, Y:=-121.4, Z:=221.4), (X:=336.3, Y:=-121.2, Z:=221.4), (X:=294.3, Y:=-121.1, Z:=221.5), (X:=252.4, Y:=-120.9, Z:=221.5),
	(X:=546.5, Y:=-79.3,  Z:=221.5), (X:=504.5, Y:=-79.1,  Z:=221.5), (X:=462.5, Y:=-78.9,  Z:=221.6), (X:=420.5, Y:=-78.7,  Z:=221.6),
	(X:=378.5, Y:=-78.4,  Z:=221.7), (X:=336.5, Y:=-78.2,  Z:=221.7), (X:=294.4, Y:=-78.0,  Z:=221.7), (X:=252.4, Y:=-77.8,  Z:=221.8),
	(X:=546.9, Y:=-36.6,  Z:=221.7), (X:=504.9, Y:=-36.3,  Z:=221.8), (X:=462.8, Y:=-36.1,  Z:=221.8), (X:=420.7, Y:=-35.8,  Z:=221.9),
	(X:=378.7, Y:=-35.5,  Z:=221.9), (X:=336.6, Y:=-35.2,  Z:=222.0), (X:=294.6, Y:=-35.0,  Z:=222.0), (X:=252.5, Y:=-34.7,  Z:=222.1),
	(X:=547.4, Y:=6.1,    Z:=222.0), (X:=505.3, Y:=6.4,    Z:=222.1), (X:=463.2, Y:=6.7,    Z:=222.1), (X:=421.0, Y:=7.1,    Z:=222.2),
	(X:=378.9, Y:=7.4,    Z:=222.2), (X:=336.8, Y:=7.8,    Z:=222.3), (X:=294.7, Y:=8.1,    Z:=222.3), (X:=252.5, Y:=8.4,    Z:=222.4),
	(X:=547.9, Y:=48.7,   Z:=222.3), (X:=505.7, Y:=49.1,   Z:=222.3), (X:=463.5, Y:=49.5,   Z:=222.4), (X:=421.3, Y:=49.9,   Z:=222.4),
	(X:=379.1, Y:=50.4,   Z:=222.5), (X:=336.9, Y:=50.8,   Z:=222.5), (X:=294.8, Y:=51.2,   Z:=222.6), (X:=252.6, Y:=51.6,   Z:=222.6),
	(X:=548.4, Y:=91.4,   Z:=222.6), (X:=506.1, Y:=91.9,   Z:=222.6), (X:=463.9, Y:=92.4,   Z:=222.7), (X:=421.6, Y:=92.8,   Z:=222.7),
	(X:=379.4, Y:=93.3,   Z:=222.8), (X:=337.1, Y:=93.7,   Z:=222.8), (X:=294.9, Y:=94.2,   Z:=222.9), (X:=252.6, Y:=94.7,   Z:=222.9),
	(X:=548.8, Y:=134.1,  Z:=222.8), (X:=506.5, Y:=134.6,  Z:=222.9), (X:=464.2, Y:=135.2,  Z:=222.9), (X:=421.9, Y:=135.7,  Z:=223.0),
	(X:=379.6, Y:=136.2,  Z:=223.0), (X:=337.3, Y:=136.7,  Z:=223.1), (X:=295.0, Y:=137.3,  Z:=223.2), (X:=252.7, Y:=137.8,  Z:=223.2),
	(X:=549.3, Y:=176.8,  Z:=223.1), (X:=506.9, Y:=177.4,  Z:=223.2), (X:=464.6, Y:=178.0,  Z:=223.2), (X:=422.2, Y:=178.6,  Z:=223.3),
	(X:=379.8, Y:=179.1,  Z:=223.3), (X:=337.4, Y:=179.7,  Z:=223.4), (X:=295.1, Y:=180.3,  Z:=223.4), (X:=252.7, Y:=180.9,  Z:=223.5)
];END_VAR
```

#### Main.st
```iecst
PROGRAM _INIT
	(* Insert code here *)
	gMotionInterface.BlackPilePos.X := 395.4;
	gMotionInterface.BlackPilePos.Y := -293;
	gMotionInterface.BlackPilePos.Z := 286.4;

	gMotionInterface.WhitePilePos.X := 395.4;
	gMotionInterface.WhitePilePos.Y := -293;
	gMotionInterface.WhitePilePos.Z := 286.4;

END_PROGRAM

PROGRAM _CYCLIC
	IF gStep = RobotMove AND gRobotMoveVar.RTRMove THEN
		CASE MoveStep OF
			IdleRM:
				MoveStep := MoveExecute;

			MoveExecute:
				IF gMotionInterface.Ready THEN
					gMotionInterface.Command := MOVE_START_END;
					gMotionInterface.StartPos := COORD_POSITION[gRobotMoveVar.StartPoint.x,gRobotMoveVar.StartPoint.y];
					gMotionInterface.EndPos := COORD_POSITION[gRobotMoveVar.EndPoint.x,gRobotMoveVar.EndPoint.y];
					gMotionInterface.Execute := TRUE;
					MoveStep := MoveBusy;
				END_IF;

			MoveBusy:
				IF gMotionInterface.Done THEN
					gMotionInterface.Execute := FALSE;
					IF gRobotMoveVar.Capture THEN
						MoveStep := DiscardExecute;
					ELSE
						MoveStep := EndRM;
					END_IF;
				END_IF;

			DiscardExecute:
				IF gMotionInterface.Ready THEN
					IF gRobotMoveVar.DiscardColorWhite THEN
						gMotionInterface.Command := DISCARD_WHITE;
					ELSE
						gMotionInterface.Command := DISCARD_BLACK;
					END_IF;
					gMotionInterface.StartPos := COORD_POSITION[gRobotMoveVar.DiscardPoint.x,gRobotMoveVar.DiscardPoint.y];
					gMotionInterface.Execute := TRUE;
					MoveStep := DiscardBusy;
				END_IF;

			DiscardBusy:
				IF gMotionInterface.Done THEN
					gMotionInterface.Execute := FALSE;
					MoveStep := EndRM;
				END_IF;

			EndRM:
				MoveStep := IdleRM;
				gStep := PhotoCheck;
				gRobotMoveVar.RTRMove := FALSE;
		END_CASE;
	END_IF;

END_PROGRAM

PROGRAM _EXIT
	(* Insert code here *)

END_PROGRAM
```

### Program Logical/Programs/Motion/RobotMovements (IEC)

#### Main.st - Init, cyclic, exit code
```iecst
PROGRAM _INIT
	FOR row := 1 TO 8 DO
		FOR col := 1 TO 8 DO
			gPositionMatrix[row, col].X := (row - 1) * 50;
			gPositionMatrix[row, col].Y := (col - 1) * 50;
			gPositionMatrix[row, col].Z := 50;
		END_FOR
	END_FOR
END_PROGRAM

PROGRAM _CYCLIC
	instRobotMove(
		PickPiece := gPickPiece,
		PickMove := gPickMove,
		PositionMatrix := gPositionMatrix,
		Motion := gMotionInterface
		);
END_PROGRAM

PROGRAM _EXIT
	(* Insert code here *)

END_PROGRAM
```

#### Variables.var - Local variables
```iecst
VAR
	col : INT;
	row : INT;
	instRobotMove : FB_MovePiece;
END_VAR
```

#### LocalFunctions.fun
```iecst
{REDUND_ERROR} {REDUND_UNREPLICABLE} FUNCTION_BLOCK FB_MovePiece (*TODO: Add your comment here*) (*$GROUP=User,$CAT=User,$GROUPICON=User.png,$CATICON=User.png*)
	VAR_INPUT
		PickPiece  : ARRAY[1..8,1..8] OF BOOL;
		PickMove   : ARRAY[1..8,1..8] OF BOOL;
		PositionMatrix : ARRAY[1..8,1..8] OF McPosType;
	END_VAR

	VAR_IN_OUT
		Motion      : MotionInterfaceType;
	END_VAR

	VAR_OUTPUT
		Done        : BOOL;
		Busy        : BOOL;
	END_VAR

	VAR
    	iState : INT := 0;
		Row : INT;
		Col : INT;
		AnyPickPiece : BOOL; (* Flaga: czy jakikolwiek pionek jest wybrany *)
		AnyPickMove : BOOL;   (* Flaga: czy jakikolwiek ruch jest wybrany *)
	END_VAR
END_FUNCTION_BLOCK
```

#### FB_MovePiece.st
```iecst
(* TODO: Add your comment here *)
FUNCTION_BLOCK FB_MovePiece

	AnyPickPiece := FALSE;
	AnyPickMove := FALSE;

	FOR Row := 1 TO 8 DO
		FOR Col := 1 TO 8 DO
			IF PickPiece[Row, Col] THEN AnyPickPiece := TRUE; END_IF;
			IF PickMove[Row, Col] THEN AnyPickMove := TRUE; END_IF;
		END_FOR;
	END_FOR;

	(* --- KROK 2: MASZYNA STANÓW --- *)
	CASE iState OF
		0: (* Oczekiwanie na sygnał od gracza *)
			(* Teraz Twoja logika: jeśli gracz wybrał pionek I cel, startujemy *)
			IF AnyPickPiece AND AnyPickMove THEN
				iState := 10;
			END_IF;
		10: (* STAN: Wyznaczenie współrzędnych *)
			FOR Row := 1 TO 8 DO
				FOR Col := 1 TO 8 DO
					IF PickPiece[Row,Col] THEN
						Motion.StartPos := PositionMatrix[Row,Col];
					END_IF;
					IF PickMove[Row,Col] THEN
						Motion.EndPos := PositionMatrix[Row,Col];
					END_IF;
				END_FOR;
			END_FOR;

			Motion.Move := TRUE; (* Wyzwalacz ruchu - tylko raz! *)
			iState := 20;

		20: (* STAN: Oczekiwanie na zakończenie ruchu *)
			IF Motion.Done THEN (* Załóżmy, że Motion ma wyjście Done *)
				Motion.Move := FALSE; (* Reset sygnału dla kolejnego ruchu *)
				iState := 30;
			END_IF;

		30: (* STAN: Reset danych silnika warcabów *)
			FOR Row := 1 TO 8 DO
				FOR Col := 1 TO 8 DO
					PickPiece[Row, Col] := FALSE;
					PickMove[Row, Col] := FALSE;
				END_FOR;
			END_FOR;
		iState := 0; (* Powrót do oczekiwania *)
	END_CASE;

	FOR Row := 1 TO 8 DO
		FOR Col := 1 TO 8 DO

			IF PickPiece[Row,Col] THEN
				Motion.StartPos := PositionMatrix[Row,Col];
			END_IF;

			IF PickMove[Row,Col] THEN
				Motion.EndPos := PositionMatrix[Row,Col];
			END_IF;

		END_FOR;
	END_FOR;

	Motion.Move := TRUE;
END_FUNCTION_BLOCK
```

### Program Logical/Programs/camera (IEC)
